// TIA Portal V19 program export: 1 tag tables, 0 data types, 4 data blocks, 12 code blocks (in call order from the OBs), 14 instance data blocks

VAR_GLOBAL   // PLC tag table "System"
   System_Byte AT %MB1 : Byte;
   FirstScan AT %M1.0 : Bool;
   DiagStatusUpdate AT %M1.1 : Bool;
   AlwaysTRUE AT %M1.2 : Bool;
   AlwaysFALSE AT %M1.3 : Bool;
   Clock_Byte AT %MB0 : Byte;
   Clock_10Hz AT %M0.0 : Bool;
   Clock_5Hz AT %M0.1 : Bool;
   "Clock_2.5Hz" AT %M0.2 : Bool;
   Clock_2Hz AT %M0.3 : Bool;
   "Clock_1.25Hz" AT %M0.4 : Bool;
   Clock_1Hz AT %M0.5 : Bool;
   "Clock_0.625Hz" AT %M0.6 : Bool;
   "Clock_0.5Hz" AT %M0.7 : Bool;
   Tag_1 AT %M10.0 : Bool;
END_VAR

DATA_BLOCK "DB_Parameters"   // DB2
{ S7_Optimized_Access := 'TRUE'; DB_Accessible_From_OPC_UA := 'FALSE' }
// stored: DBAccessibleFromOPCUA false, DBAccessibleFromWebserver false, MemoryReserve 100
   VAR RETAIN
      SensorParameter42B4 { ExternalAccessible := 'False'; ExternalVisible := 'False'; ExternalWritable := 'False'} : "stConfigScaleIntReal";   // Parameter for sensor car body detection (42B4 & 42B3)
      SwitchSensorValue { ExternalAccessible := 'False'; ExternalVisible := 'False'; ExternalWritable := 'False'} : Real := 650.0;   // Level parameter switch for car body detection
      uiSpeedLockEccentric { ExternalAccessible := 'False'; ExternalVisible := 'False'; ExternalWritable := 'False'} : UInt := 50;   // Rotation speed for lock eccentric
      RemoveSandPaperParam { ExternalAccessible := 'False'; ExternalVisible := 'False'; ExternalWritable := 'False'} : "stFerRoboticParam";   // FerRobotic parameter for remove the wor sandpaper
      PickUpSandPaperParam { ExternalAccessible := 'False'; ExternalVisible := 'False'; ExternalWritable := 'False'} : "stFerRoboticParam";   // FerRobotic parameter for pich up a new sandpaper
      FlatnessCtrlParam { ExternalAccessible := 'False'; ExternalVisible := 'False'; ExternalWritable := 'False'} : "stFerRoboticParam";   // FerRobotic paramter for flatness contrl disk planeity
      ConfigGreaseZaxis { ExternalAccessible := 'False'; ExternalVisible := 'False'; ExternalWritable := 'False'} : "stConfigGrease";
      ConfigGreaseXaxis { ExternalAccessible := 'False'; ExternalVisible := 'False'; ExternalWritable := 'False'} : "stConfigGrease";
      ConfigVacuumValve { ExternalAccessible := 'False'; ExternalVisible := 'False'; ExternalWritable := 'False'} : "stConfigActuator";
      tTimeoutGimball { ExternalAccessible := 'False'; ExternalVisible := 'False'; ExternalWritable := 'False'} : Time := T#5S;
      tTimeoutEccentric { ExternalAccessible := 'False'; ExternalVisible := 'False'; ExternalWritable := 'False'} : Time := T#20S;
      rFlatnessStrockPos { ExternalAccessible := 'False'; ExternalVisible := 'False'; ExternalWritable := 'False'} : Real := 23.9;   // FerRobotic strock position for control flatness
      rDeltaFlatnessStrock { ExternalAccessible := 'False'; ExternalVisible := 'False'; ExternalWritable := 'False'} : Real := 0.8;   // Delta maxi for flatness control
      nNbDiskLeft { ExternalAccessible := 'False'; ExternalVisible := 'False'; ExternalWritable := 'False'} : USInt := 2;
      nNbDiskRight { ExternalAccessible := 'False'; ExternalVisible := 'False'; ExternalWritable := 'False'} : USInt := 1;
      rLowLimiteStroke { ExternalAccessible := 'False'; ExternalVisible := 'False'; ExternalWritable := 'False'} : Real := 5.0;
      StrokeTooExtend { ExternalAccessible := 'False'; ExternalVisible := 'False'; ExternalWritable := 'False'} : "stHysteresis";
      StrokeTooRetract { ExternalAccessible := 'False'; ExternalVisible := 'False'; ExternalWritable := 'False'} : "stHysteresis";
   END_VAR
BEGIN
   SensorParameter42B4.nInputMin := 0;
   SensorParameter42B4.nIntputMax := 27648;
   SensorParameter42B4.xUniPolar := TRUE;
   SensorParameter42B4.xReverseValue := TRUE;
   SensorParameter42B4.rOutputMin := 200.0;
   SensorParameter42B4.rOutputMax := 1000.0;
   SensorParameter42B4.rOffsetFixe := 0.0;
   SensorParameter42B4.rOffsetProp := 1.0;
   RemoveSandPaperParam.nSetForceTarget := 20;
   RemoveSandPaperParam.nSetForceZero := 10;
   RemoveSandPaperParam.usiSetTimeRamp := 0;
   RemoveSandPaperParam.uiSetSpeed := 0;
   PickUpSandPaperParam.nSetForceTarget := 100;
   PickUpSandPaperParam.nSetForceZero := 0;
   PickUpSandPaperParam.usiSetTimeRamp := 0;
   PickUpSandPaperParam.uiSetSpeed := 0;
   FlatnessCtrlParam.nSetForceTarget := 20;
   FlatnessCtrlParam.nSetForceZero := 0;
   FlatnessCtrlParam.usiSetTimeRamp := 0;
   FlatnessCtrlParam.uiSetSpeed := 0;
   ConfigGreaseZaxis.uiNbPulsePerKm := 4411;
   ConfigGreaseZaxis.uiKmForGreasing := 32;
   ConfigGreaseZaxis.tTimeEnableGreasePump := T#1M;
   ConfigGreaseZaxis.tTimeoutPxGrease := T#1M;
   ConfigGreaseXaxis.uiNbPulsePerKm := 4411;
   ConfigGreaseXaxis.uiKmForGreasing := 32;
   ConfigGreaseXaxis.tTimeEnableGreasePump := T#2M;
   ConfigGreaseXaxis.tTimeoutPxGrease := T#2M;
   ConfigVacuumValve.xEnaMeasureTimeHome := FALSE;
   ConfigVacuumValve.xEnaMeasureTimeAction := FALSE;
   ConfigVacuumValve.xKeepHomeSolActive := FALSE;
   ConfigVacuumValve.xKeepActionSolActive := TRUE;
   ConfigVacuumValve.xPresHomePxSensor := TRUE;
   ConfigVacuumValve.xPresActionPxSensor := TRUE;
   ConfigVacuumValve.tSwitchingCommand := T#50MS;
   ConfigVacuumValve.tTimeOutHomeSensor := T#8S;
   ConfigVacuumValve.tTimeOutActionSensor := T#8S;
   ConfigVacuumValve.tHomeTime := T#3S;
   ConfigVacuumValve.tActionTime := T#3S;
   ConfigVacuumValve.tFilterPxHome := T#100MS;
   ConfigVacuumValve.tFilterPxAction := T#100MS;
   StrokeTooExtend.rValueOn := 40.0;
   StrokeTooExtend.rValueOff := 35.0;
   StrokeTooRetract.rValueOn := 8.0;
   StrokeTooRetract.rValueOff := 13.0;
END_DATA_BLOCK

DATA_BLOCK "DB_Fault"   // DB90
{ S7_Optimized_Access := 'TRUE'; DB_Accessible_From_OPC_UA := 'FALSE' }
// stored: AutoNumber false, DBAccessibleFromOPCUA false, DBAccessibleFromWebserver false, MemoryReserve 100
   VAR
      tonFeedbackZAxisError { ExternalAccessible := 'False'; ExternalVisible := 'False'; ExternalWritable := 'False'} : TON_TIME;
      tonFautLockZAxis { ExternalAccessible := 'False'; ExternalVisible := 'False'; ExternalWritable := 'False'} : TON_TIME;
      tonFaultUnlockZAxis { ExternalAccessible := 'False'; ExternalVisible := 'False'; ExternalWritable := 'False'} : TON_TIME;
      tonFaultStrokTooRetracted { ExternalAccessible := 'False'; ExternalVisible := 'False'; ExternalWritable := 'False'} : TON_TIME;
   END_VAR
BEGIN
END_DATA_BLOCK

DATA_BLOCK "DBF_Safety"   // DB901, F_DB
{ S7_Optimized_Access := 'TRUE' }
// stored: AutoNumber false
   VAR
      TrueSafety { ExternalAccessible := 'False'; ExternalVisible := 'False'; ExternalWritable := 'False'} : Bool := TRUE;   // Bit de securite toujours vrai
      FalseSafety { ExternalAccessible := 'False'; ExternalVisible := 'False'; ExternalWritable := 'False'} : Bool := FALSE;   // Bit de securite toujours faux
      Reset { ExternalAccessible := 'False'; ExternalVisible := 'False'; ExternalWritable := 'False'} : Bool;   // Bit de reset
      i_FdbZAxisBrake { ExternalAccessible := 'False'; ExternalVisible := 'False'; ExternalWritable := 'False'} : Bool;   // Feedback solenoid valve
      i_ResetFromMaster { ExternalAccessible := 'False'; ExternalVisible := 'False'; ExternalWritable := 'False'} : Bool;   // Reset safety from Master PLC
      i_EStopFromMaster { ExternalAccessible := 'False'; ExternalVisible := 'False'; ExternalWritable := 'False'} : Bool;   // Emergency stop from master PLC
      i_OProtectFromMaster { ExternalAccessible := 'False'; ExternalVisible := 'False'; ExternalWritable := 'False'} : Bool;   // Operator Protection from master PLC
      i_AirSupplyEnabledFromMaster { ExternalAccessible := 'False'; ExternalVisible := 'False'; ExternalWritable := 'False'} : Bool;   // Air pressure enabled from master PLC
      i_StopStrokeLimit { ExternalAccessible := 'False'; ExternalVisible := 'False'; ExternalWritable := 'False'} : Bool;   // Stop Stroke limite
      i_VacuumPumpRunning { ExternalAccessible := 'False'; ExternalVisible := 'False'; ExternalWritable := 'False'} : Bool;   // Vacuum pump is running - Zero Speed detection
      o_UnlockZAxis { ExternalAccessible := 'False'; ExternalVisible := 'False'; ExternalWritable := 'False'} : Bool;   // Unlock Z axis of robot
      o_SafetyEnable { ExternalAccessible := 'False'; ExternalVisible := 'False'; ExternalWritable := 'False'} : Bool;   // Safety enabled to Robot Safemove
      o_ExternalEStopToRobot { ExternalAccessible := 'False'; ExternalVisible := 'False'; ExternalWritable := 'False'} : Bool;   // External emergency stop to Robot Safemove
      o_ExternalOProtectToRobot { ExternalAccessible := 'False'; ExternalVisible := 'False'; ExternalWritable := 'False'} : Bool;   // External operator protection to robot Safemove
      o_EStoptoMaster { ExternalAccessible := 'False'; ExternalVisible := 'False'; ExternalWritable := 'False'} : Bool;   // Internal Emergency stop to master PLC
      o_ReqAirSupplyToMaster { ExternalAccessible := 'False'; ExternalVisible := 'False'; ExternalWritable := 'False'} : Bool;   // Request enable air pressure supply to master PLC
      o_RobotStopperToMaster { ExternalAccessible := 'False'; ExternalVisible := 'False'; ExternalWritable := 'False'} : Bool;   // Robot stopped state to master PLC
      o_PowerOffFerRobotic { ExternalAccessible := 'False'; ExternalVisible := 'False'; ExternalWritable := 'False'} : Bool;   // Power Off 24V Safety for FerRobotic
      xErrorReadFromMaster { ExternalAccessible := 'False'; ExternalVisible := 'False'; ExternalWritable := 'False'} : Bool;   // Error read safety data from Master PLC
      xErrorWriteToMaster { ExternalAccessible := 'False'; ExternalVisible := 'False'; ExternalWritable := 'False'} : Bool;   // Error write safety data to Master PLC
   END_VAR
BEGIN
END_DATA_BLOCK

DATA_BLOCK "DB_ToSafety"   // DB999
{ S7_Optimized_Access := 'TRUE' }
// stored: AutoNumber false, MemoryReserve 100
   VAR
      xReset { ExternalAccessible := 'False'; ExternalVisible := 'False'; ExternalWritable := 'False'} : Bool;   // Commande reset general
      xStopStrokeLimit { ExternalAccessible := 'False'; ExternalVisible := 'False'; ExternalWritable := 'False'} : Bool;   // Stop robot on stroke limit retracted
      xSemiAutomaticMode { ExternalAccessible := 'False'; ExternalVisible := 'False'; ExternalWritable := 'False'} : Bool;
   END_VAR
BEGIN
END_DATA_BLOCK

ORGANIZATION_BLOCK "Main"   // OB1, LAD, ProgramCycle
TITLE = "Main Program Sweep (Cycle)"
{ S7_Optimized_Access := 'TRUE' }
// stored: SetENOAutomatically false
   VAR_INPUT
      Initial_Call : Bool;   // Initial call of this OB
      Remanence : Bool;   // =True, if remanent data are available
   END_VAR
BEGIN

REGION Network 1: Commande reset general
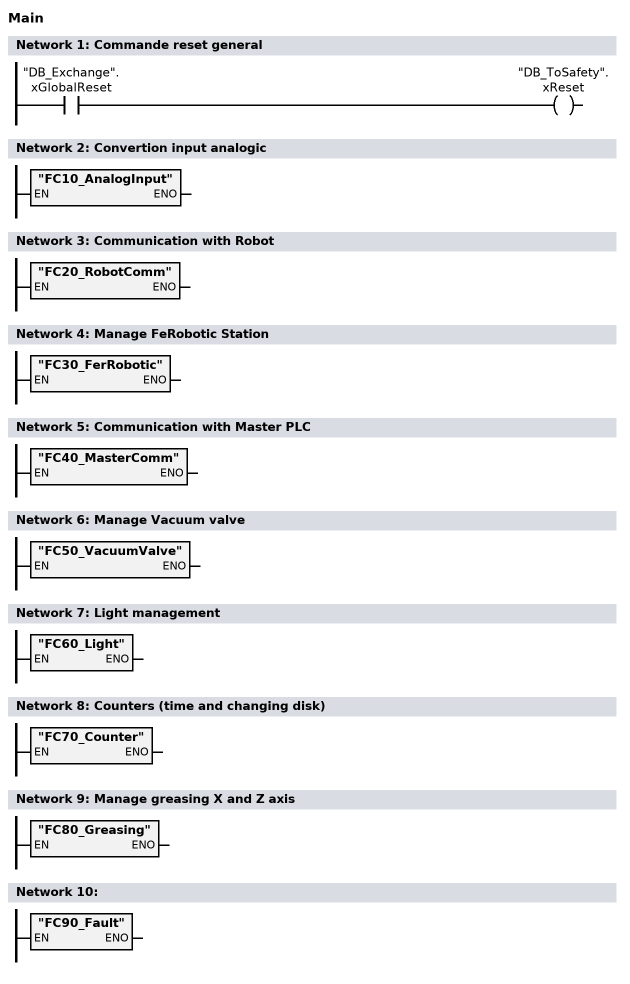
   RUNG wire#powerrail
      Contact( "DB_Exchange".xGlobalReset )
      Coil( "DB_ToSafety".xReset )
   END_RUNG
   // the same network as SCL:
   "DB_ToSafety".xReset := "DB_Exchange".xGlobalReset;
END_REGION

REGION Network 2: Convertion input analogic
   RUNG wire#powerrail
      "FC10_AnalogInput"()
   END_RUNG
   // the same network as SCL:
   "FC10_AnalogInput"();
END_REGION

REGION Network 3: Communication with Robot
   RUNG wire#powerrail
      "FC20_RobotComm"()
   END_RUNG
   // the same network as SCL:
   "FC20_RobotComm"();
END_REGION

REGION Network 4: Manage FeRobotic Station
   RUNG wire#powerrail
      "FC30_FerRobotic"()
   END_RUNG
   // the same network as SCL:
   "FC30_FerRobotic"();
END_REGION

REGION Network 5: Communication with Master PLC
   RUNG wire#powerrail
      "FC40_MasterComm"()
   END_RUNG
   // the same network as SCL:
   "FC40_MasterComm"();
END_REGION

REGION Network 6: Manage Vacuum valve
   RUNG wire#powerrail
      "FC50_VacuumValve"()
   END_RUNG
   // the same network as SCL:
   "FC50_VacuumValve"();
END_REGION

REGION Network 7: Light management
   RUNG wire#powerrail
      "FC60_Light"()
   END_RUNG
   // the same network as SCL:
   "FC60_Light"();
END_REGION

REGION Network 8: Counters (time and changing disk)
   RUNG wire#powerrail
      "FC70_Counter"()
   END_RUNG
   // the same network as SCL:
   "FC70_Counter"();
END_REGION

REGION Network 9: Manage greasing X and Z axis
   RUNG wire#powerrail
      "FC80_Greasing"()
   END_RUNG
   // the same network as SCL:
   "FC80_Greasing"();
END_REGION

REGION Network 10
   RUNG wire#powerrail
      "FC90_Fault"()
   END_RUNG
   // the same network as SCL:
   "FC90_Fault"();
END_REGION
END_ORGANIZATION_BLOCK

FUNCTION "FC30_FerRobotic" : Void   // FC30, LAD
TITLE = FerRobotic communication
{ S7_Optimized_Access := 'TRUE' }
// stored: AutoNumber false, IsIECCheckEnabled true, SetENOAutomatically false
BEGIN

REGION Network 1: Swap byte of value to Receive from FerRobotic
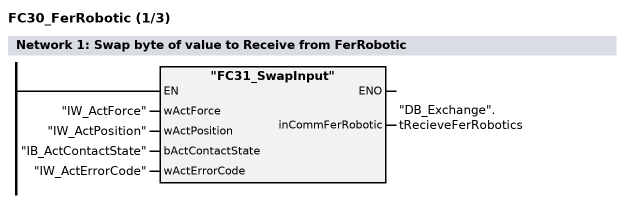
   RUNG wire#powerrail
      "FC31_SwapInput"(wActForce := "IW_ActForce", wActPosition := "IW_ActPosition", bActContactState := "IB_ActContactState", wActErrorCode := "IW_ActErrorCode", inCommFerRobotic => "DB_Exchange".tRecieveFerRobotics)
   END_RUNG
   // the same network as SCL:
   "FC31_SwapInput"(wActForce := "IW_ActForce",
                    wActPosition := "IW_ActPosition",
                    bActContactState := "IB_ActContactState",
                    wActErrorCode := "IW_ActErrorCode",
                    inCommFerRobotic => "DB_Exchange".tRecieveFerRobotics);
END_REGION

REGION Network 2: Comminucation with FerRobotic System
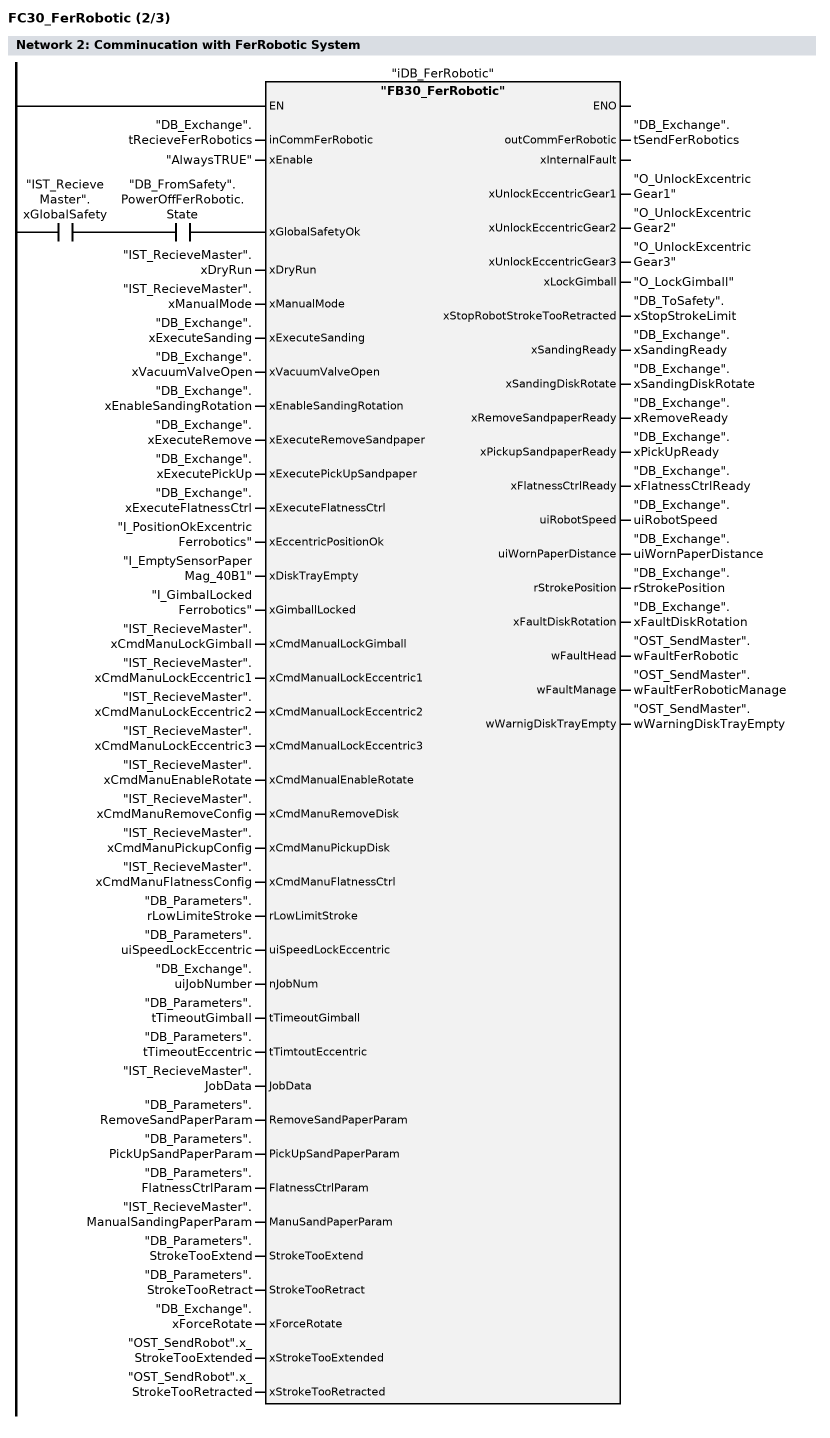
   RUNG wire#powerrail
      "iDB_FerRobotic"(xGlobalSafetyOk := wire#w1, inCommFerRobotic := "DB_Exchange".tRecieveFerRobotics, xEnable := "AlwaysTRUE", xDryRun := "IST_RecieveMaster".xDryRun, xManualMode := "IST_RecieveMaster".xManualMode, xExecuteSanding := "DB_Exchange".xExecuteSanding, xVacuumValveOpen := "DB_Exchange".xVacuumValveOpen, xEnableSandingRotation := "DB_Exchange".xEnableSandingRotation, xExecuteRemoveSandpaper := "DB_Exchange".xExecuteRemove, xExecutePickUpSandpaper := "DB_Exchange".xExecutePickUp, xExecuteFlatnessCtrl := "DB_Exchange".xExecuteFlatnessCtrl, xEccentricPositionOk := "I_PositionOkExcentricFerrobotics", xDiskTrayEmpty := "I_EmptySensorPaperMag_40B1", xGimballLocked := "I_GimbalLockedFerrobotics", xCmdManualLockGimball := "IST_RecieveMaster".xCmdManuLockGimball, xCmdManualLockEccentric1 := "IST_RecieveMaster".xCmdManuLockEccentric1, xCmdManualLockEccentric2 := "IST_RecieveMaster".xCmdManuLockEccentric2, xCmdManualLockEccentric3 := "IST_RecieveMaster".xCmdManuLockEccentric3, xCmdManualEnableRotate := "IST_RecieveMaster".xCmdManuEnableRotate, xCmdManuRemoveDisk := "IST_RecieveMaster".xCmdManuRemoveConfig, xCmdManuPickupDisk := "IST_RecieveMaster".xCmdManuPickupConfig, xCmdManuFlatnessCtrl := "IST_RecieveMaster".xCmdManuFlatnessConfig, rLowLimitStroke := "DB_Parameters".rLowLimiteStroke, uiSpeedLockEccentric := "DB_Parameters".uiSpeedLockEccentric, nJobNum := "DB_Exchange".uiJobNumber, tTimeoutGimball := "DB_Parameters".tTimeoutGimball, tTimtoutEccentric := "DB_Parameters".tTimeoutEccentric, JobData := "IST_RecieveMaster".JobData, RemoveSandPaperParam := "DB_Parameters".RemoveSandPaperParam, PickUpSandPaperParam := "DB_Parameters".PickUpSandPaperParam, FlatnessCtrlParam := "DB_Parameters".FlatnessCtrlParam, ManuSandPaperParam := "IST_RecieveMaster".ManualSandingPaperParam, StrokeTooExtend := "DB_Parameters".StrokeTooExtend, StrokeTooRetract := "DB_Parameters".StrokeTooRetract, xForceRotate := "DB_Exchange".xForceRotate, xStrokeTooExtended := "OST_SendRobot".x_StrokeTooExtended, xStrokeTooRetracted := "OST_SendRobot".x_StrokeTooRetracted, outCommFerRobotic => "DB_Exchange".tSendFerRobotics, xInternalFault =>, xUnlockEccentricGear1 => "O_UnlockExcentricGear1", xUnlockEccentricGear2 => "O_UnlockExcentricGear2", xUnlockEccentricGear3 => "O_UnlockExcentricGear3", xLockGimball => "O_LockGimball", xStopRobotStrokeTooRetracted => "DB_ToSafety".xStopStrokeLimit, xSandingReady => "DB_Exchange".xSandingReady, xSandingDiskRotate => "DB_Exchange".xSandingDiskRotate, xRemoveSandpaperReady => "DB_Exchange".xRemoveReady, xPickupSandpaperReady => "DB_Exchange".xPickUpReady, xFlatnessCtrlReady => "DB_Exchange".xFlatnessCtrlReady, uiRobotSpeed => "DB_Exchange".uiRobotSpeed, uiWornPaperDistance => "DB_Exchange".uiWornPaperDistance, rStrokePosition => "DB_Exchange".rStrokePosition, xFaultDiskRotation => "DB_Exchange".xFaultDiskRotation, wFaultHead => "OST_SendMaster".wFaultFerRobotic, wFaultManage => "OST_SendMaster".wFaultFerRoboticManage, wWarnigDiskTrayEmpty => "OST_SendMaster".wWarningDiskTrayEmpty)
   END_RUNG
   RUNG wire#powerrail
      Contact( "IST_RecieveMaster".xGlobalSafety )
      Contact( "DB_FromSafety".PowerOffFerRobotic.State )
   END_RUNG wire#w1
   // the same network as SCL:
   "iDB_FerRobotic"(inCommFerRobotic := "DB_Exchange".tRecieveFerRobotics,   // "FB30_FerRobotic"
                    xEnable := "AlwaysTRUE",
                    xGlobalSafetyOk := "IST_RecieveMaster".xGlobalSafety AND "DB_FromSafety".PowerOffFerRobotic.State,
                    xDryRun := "IST_RecieveMaster".xDryRun,
                    xManualMode := "IST_RecieveMaster".xManualMode,
                    xExecuteSanding := "DB_Exchange".xExecuteSanding,
                    xVacuumValveOpen := "DB_Exchange".xVacuumValveOpen,
                    xEnableSandingRotation := "DB_Exchange".xEnableSandingRotation,
                    xExecuteRemoveSandpaper := "DB_Exchange".xExecuteRemove,
                    xExecutePickUpSandpaper := "DB_Exchange".xExecutePickUp,
                    xExecuteFlatnessCtrl := "DB_Exchange".xExecuteFlatnessCtrl,
                    xEccentricPositionOk := "I_PositionOkExcentricFerrobotics",
                    xDiskTrayEmpty := "I_EmptySensorPaperMag_40B1",
                    xGimballLocked := "I_GimbalLockedFerrobotics",
                    xCmdManualLockGimball := "IST_RecieveMaster".xCmdManuLockGimball,
                    xCmdManualLockEccentric1 := "IST_RecieveMaster".xCmdManuLockEccentric1,
                    xCmdManualLockEccentric2 := "IST_RecieveMaster".xCmdManuLockEccentric2,
                    xCmdManualLockEccentric3 := "IST_RecieveMaster".xCmdManuLockEccentric3,
                    xCmdManualEnableRotate := "IST_RecieveMaster".xCmdManuEnableRotate,
                    xCmdManuRemoveDisk := "IST_RecieveMaster".xCmdManuRemoveConfig,
                    xCmdManuPickupDisk := "IST_RecieveMaster".xCmdManuPickupConfig,
                    xCmdManuFlatnessCtrl := "IST_RecieveMaster".xCmdManuFlatnessConfig,
                    rLowLimitStroke := "DB_Parameters".rLowLimiteStroke,
                    uiSpeedLockEccentric := "DB_Parameters".uiSpeedLockEccentric,
                    nJobNum := "DB_Exchange".uiJobNumber,
                    tTimeoutGimball := "DB_Parameters".tTimeoutGimball,
                    tTimtoutEccentric := "DB_Parameters".tTimeoutEccentric,
                    JobData := "IST_RecieveMaster".JobData,
                    RemoveSandPaperParam := "DB_Parameters".RemoveSandPaperParam,
                    PickUpSandPaperParam := "DB_Parameters".PickUpSandPaperParam,
                    FlatnessCtrlParam := "DB_Parameters".FlatnessCtrlParam,
                    ManuSandPaperParam := "IST_RecieveMaster".ManualSandingPaperParam,
                    StrokeTooExtend := "DB_Parameters".StrokeTooExtend,
                    StrokeTooRetract := "DB_Parameters".StrokeTooRetract,
                    xForceRotate := "DB_Exchange".xForceRotate,
                    xStrokeTooExtended := "OST_SendRobot".x_StrokeTooExtended,
                    xStrokeTooRetracted := "OST_SendRobot".x_StrokeTooRetracted,
                    outCommFerRobotic => "DB_Exchange".tSendFerRobotics,
                    xUnlockEccentricGear1 => "O_UnlockExcentricGear1",
                    xUnlockEccentricGear2 => "O_UnlockExcentricGear2",
                    xUnlockEccentricGear3 => "O_UnlockExcentricGear3",
                    xLockGimball => "O_LockGimball",
                    xStopRobotStrokeTooRetracted => "DB_ToSafety".xStopStrokeLimit,
                    xSandingReady => "DB_Exchange".xSandingReady,
                    xSandingDiskRotate => "DB_Exchange".xSandingDiskRotate,
                    xRemoveSandpaperReady => "DB_Exchange".xRemoveReady,
                    xPickupSandpaperReady => "DB_Exchange".xPickUpReady,
                    xFlatnessCtrlReady => "DB_Exchange".xFlatnessCtrlReady,
                    uiRobotSpeed => "DB_Exchange".uiRobotSpeed,
                    uiWornPaperDistance => "DB_Exchange".uiWornPaperDistance,
                    rStrokePosition => "DB_Exchange".rStrokePosition,
                    xFaultDiskRotation => "DB_Exchange".xFaultDiskRotation,
                    wFaultHead => "OST_SendMaster".wFaultFerRobotic,
                    wFaultManage => "OST_SendMaster".wFaultFerRoboticManage,
                    wWarnigDiskTrayEmpty => "OST_SendMaster".wWarningDiskTrayEmpty);
END_REGION

REGION Network 3: Swap byte of value to send to FerRobotic
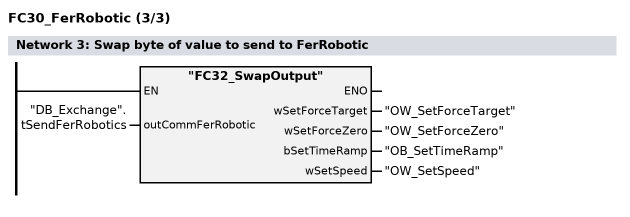
   RUNG wire#powerrail
      "FC32_SwapOutput"(outCommFerRobotic := "DB_Exchange".tSendFerRobotics, wSetForceTarget => "OW_SetForceTarget", wSetForceZero => "OW_SetForceZero", bSetTimeRamp => "OB_SetTimeRamp", wSetSpeed => "OW_SetSpeed")
   END_RUNG
   // the same network as SCL:
   "FC32_SwapOutput"(outCommFerRobotic := "DB_Exchange".tSendFerRobotics,
                     wSetForceTarget => "OW_SetForceTarget",
                     wSetForceZero => "OW_SetForceZero",
                     bSetTimeRamp => "OB_SetTimeRamp",
                     wSetSpeed => "OW_SetSpeed");
END_REGION
END_FUNCTION

FUNCTION "FC31_SwapInput" : Void
{ S7_Optimized_Access := 'TRUE' }
VERSION : 0.1
   VAR_INPUT 
      wActForce : Word;
      wActPosition : Word;
      bActContactState : Byte;
      wActErrorCode : Word;
   END_VAR

   VAR_OUTPUT 
      inCommFerRobotic : "stRecieveFerRobotics";
   END_VAR


BEGIN
	// Swap word of Act Force value
	#inCommFerRobotic.nActForce := WORD_TO_INT( SWAP(#wActForce));
	// Swap word of ActError code value
	#inCommFerRobotic.uiActErrorCode := WORD_TO_UINT(SWAP(#wActErrorCode));
	// Swap word of Act position value
	#inCommFerRobotic.uiActPosition := WORD_TO_UINT(SWAP(#wActPosition));
	// Convert Usint to word of contact state
	#inCommFerRobotic.usiActContactState := BYTE_TO_USINT(#bActContactState);
	
END_FUNCTION

FUNCTION "FC32_SwapOutput" : Void
{ S7_Optimized_Access := 'TRUE' }
VERSION : 0.1
   VAR_INPUT 
      outCommFerRobotic : "stSendFerRobotics";
   END_VAR

   VAR_OUTPUT 
      wSetForceTarget : Word;
      wSetForceZero : Word;
      bSetTimeRamp : Byte;
      wSetSpeed : Word;
   END_VAR


BEGIN
	// Swap word of Set Force Target value
	#wSetForceTarget := SWAP(INT_TO_WORD(#outCommFerRobotic.nSetForceTarget));
	// Swap word of Set Force Zero value
	#wSetForceZero := SWAP(INT_TO_WORD(#outCommFerRobotic.nSetForceZero));
	// Swap word of Set Speed value
	#wSetSpeed := SWAP(UINT_TO_WORD(#outCommFerRobotic.uiSetSpeed));
	// Convert word to USint for time Ramp value
	#bSetTimeRamp := USINT_TO_BYTE(#outCommFerRobotic.usiSetTimeRamp);
	
END_FUNCTION

FUNCTION "FC40_MasterComm" : Void   // FC40, LAD
{ S7_Optimized_Access := 'TRUE' }
// stored: AutoNumber false, IsIECCheckEnabled true, SetENOAutomatically true
BEGIN

REGION Network 1: Master Communication
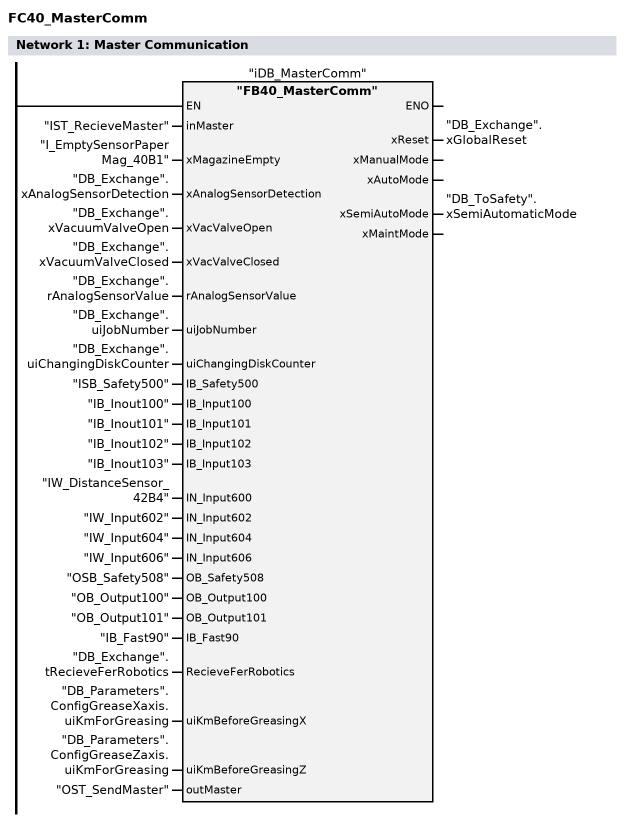
   RUNG wire#powerrail
      "iDB_MasterComm"(inMaster := "IST_RecieveMaster", xMagazineEmpty := "I_EmptySensorPaperMag_40B1", xAnalogSensorDetection := "DB_Exchange".xAnalogSensorDetection, xVacValveOpen := "DB_Exchange".xVacuumValveOpen, xVacValveClosed := "DB_Exchange".xVacuumValveClosed, rAnalogSensorValue := "DB_Exchange".rAnalogSensorValue, uiJobNumber := "DB_Exchange".uiJobNumber, uiChangingDiskCounter := "DB_Exchange".uiChangingDiskCounter, IB_Safety500 := "ISB_Safety500", IB_Input100 := "IB_Inout100", IB_Input101 := "IB_Inout101", IB_Input102 := "IB_Inout102", IB_Input103 := "IB_Inout103", IN_Input600 := "IW_DistanceSensor_42B4", IN_Input602 := "IW_Input602", IN_Input604 := "IW_Input604", IN_Input606 := "IW_Input606", OB_Safety508 := "OSB_Safety508", OB_Output100 := "OB_Output100", OB_Output101 := "OB_Output101", IB_Fast90 := "IB_Fast90", RecieveFerRobotics := "DB_Exchange".tRecieveFerRobotics, uiKmBeforeGreasingX := "DB_Parameters".ConfigGreaseXaxis.uiKmForGreasing, uiKmBeforeGreasingZ := "DB_Parameters".ConfigGreaseZaxis.uiKmForGreasing, outMaster := "OST_SendMaster", xReset => "DB_Exchange".xGlobalReset, xManualMode =>, xAutoMode =>, xSemiAutoMode => "DB_ToSafety".xSemiAutomaticMode, xMaintMode =>)
   END_RUNG
   // the same network as SCL:
   "iDB_MasterComm"(inMaster := "IST_RecieveMaster",   // "FB40_MasterComm"
                    xMagazineEmpty := "I_EmptySensorPaperMag_40B1",
                    xAnalogSensorDetection := "DB_Exchange".xAnalogSensorDetection,
                    xVacValveOpen := "DB_Exchange".xVacuumValveOpen,
                    xVacValveClosed := "DB_Exchange".xVacuumValveClosed,
                    rAnalogSensorValue := "DB_Exchange".rAnalogSensorValue,
                    uiJobNumber := "DB_Exchange".uiJobNumber,
                    uiChangingDiskCounter := "DB_Exchange".uiChangingDiskCounter,
                    IB_Safety500 := "ISB_Safety500",
                    IB_Input100 := "IB_Inout100",
                    IB_Input101 := "IB_Inout101",
                    IB_Input102 := "IB_Inout102",
                    IB_Input103 := "IB_Inout103",
                    IN_Input600 := "IW_DistanceSensor_42B4",
                    IN_Input602 := "IW_Input602",
                    IN_Input604 := "IW_Input604",
                    IN_Input606 := "IW_Input606",
                    OB_Safety508 := "OSB_Safety508",
                    OB_Output100 := "OB_Output100",
                    OB_Output101 := "OB_Output101",
                    IB_Fast90 := "IB_Fast90",
                    RecieveFerRobotics := "DB_Exchange".tRecieveFerRobotics,
                    uiKmBeforeGreasingX := "DB_Parameters".ConfigGreaseXaxis.uiKmForGreasing,
                    uiKmBeforeGreasingZ := "DB_Parameters".ConfigGreaseZaxis.uiKmForGreasing,
                    outMaster := "OST_SendMaster",
                    xReset => "DB_Exchange".xGlobalReset,
                    xSemiAutoMode => "DB_ToSafety".xSemiAutomaticMode);
END_REGION
END_FUNCTION

FUNCTION "FC70_Counter" : Void   // FC2, LAD
{ S7_Optimized_Access := 'TRUE' }
// stored: IsIECCheckEnabled true, SetENOAutomatically false
BEGIN

REGION Network 1: Running time counter
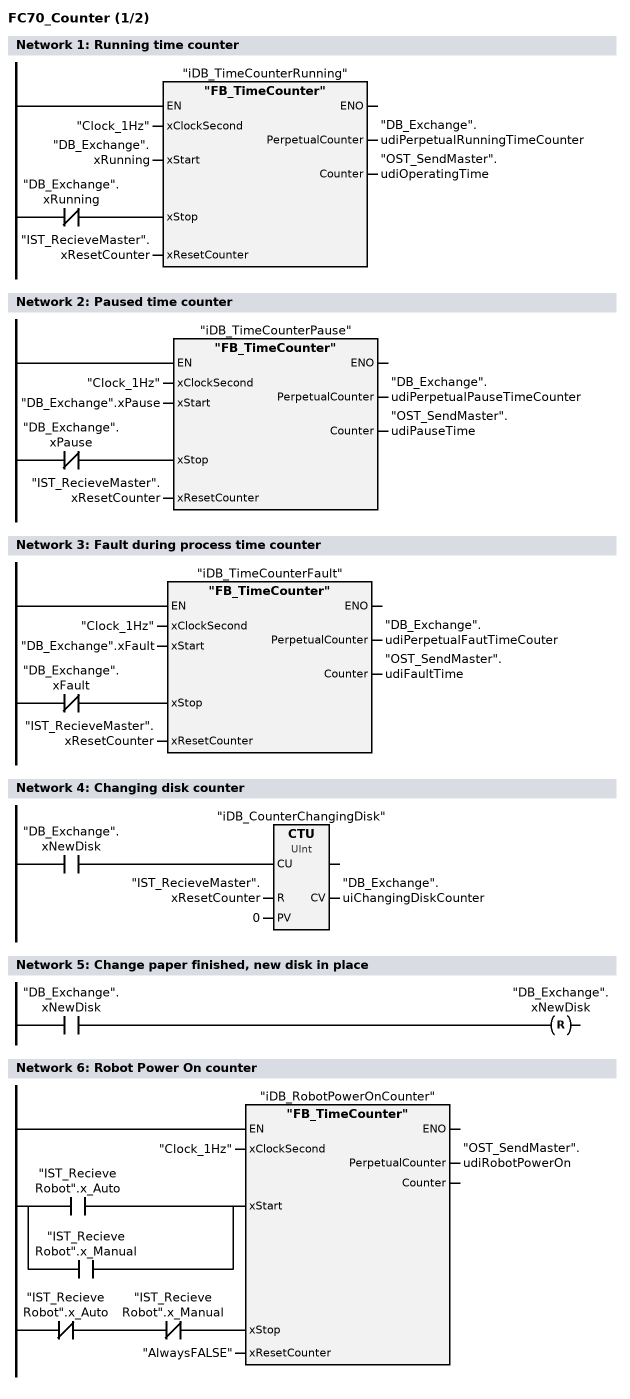
   RUNG wire#powerrail
      "iDB_TimeCounterRunning"(xStop := wire#w1, xClockSecond := "Clock_1Hz", xStart := "DB_Exchange".xRunning, xResetCounter := "IST_RecieveMaster".xResetCounter, PerpetualCounter => "DB_Exchange".udiPerpetualRunningTimeCounter, "Counter" => "OST_SendMaster".udiOperatingTime)
   END_RUNG
   RUNG wire#powerrail
      I_Contact( "DB_Exchange".xRunning )
   END_RUNG wire#w1
   // the same network as SCL:
   "iDB_TimeCounterRunning"(xClockSecond := "Clock_1Hz",   // "FB_TimeCounter"
                           xStart := "DB_Exchange".xRunning,
                           xStop := NOT "DB_Exchange".xRunning,
                           xResetCounter := "IST_RecieveMaster".xResetCounter,
                           PerpetualCounter => "DB_Exchange".udiPerpetualRunningTimeCounter,
                           "Counter" => "OST_SendMaster".udiOperatingTime);
END_REGION

REGION Network 2: Paused time counter
   RUNG wire#powerrail
      "iDB_TimeCounterPause"(xStop := wire#w1, xClockSecond := "Clock_1Hz", xStart := "DB_Exchange".xPause, xResetCounter := "IST_RecieveMaster".xResetCounter, PerpetualCounter => "DB_Exchange".udiPerpetualPauseTimeCounter, "Counter" => "OST_SendMaster".udiPauseTime)
   END_RUNG
   RUNG wire#powerrail
      I_Contact( "DB_Exchange".xPause )
   END_RUNG wire#w1
   // the same network as SCL:
   "iDB_TimeCounterPause"(xClockSecond := "Clock_1Hz",   // "FB_TimeCounter"
                          xStart := "DB_Exchange".xPause,
                          xStop := NOT "DB_Exchange".xPause,
                          xResetCounter := "IST_RecieveMaster".xResetCounter,
                          PerpetualCounter => "DB_Exchange".udiPerpetualPauseTimeCounter,
                          "Counter" => "OST_SendMaster".udiPauseTime);
END_REGION

REGION Network 3: Fault during process time counter
   RUNG wire#powerrail
      "iDB_TimeCounterFault"(xStop := wire#w1, xClockSecond := "Clock_1Hz", xStart := "DB_Exchange".xFault, xResetCounter := "IST_RecieveMaster".xResetCounter, PerpetualCounter => "DB_Exchange".udiPerpetualFautTimeCouter, "Counter" => "OST_SendMaster".udiFaultTime)
   END_RUNG
   RUNG wire#powerrail
      I_Contact( "DB_Exchange".xFault )
   END_RUNG wire#w1
   // the same network as SCL:
   "iDB_TimeCounterFault"(xClockSecond := "Clock_1Hz",   // "FB_TimeCounter"
                          xStart := "DB_Exchange".xFault,
                          xStop := NOT "DB_Exchange".xFault,
                          xResetCounter := "IST_RecieveMaster".xResetCounter,
                          PerpetualCounter => "DB_Exchange".udiPerpetualFautTimeCouter,
                          "Counter" => "OST_SendMaster".udiFaultTime);
END_REGION

REGION Network 4: Changing disk counter
   RUNG wire#powerrail
      Contact( "DB_Exchange".xNewDisk )
      { S7_Templates := "value_type := UInt" } "iDB_CounterChangingDisk".CTU(r := "IST_RecieveMaster".xResetCounter, pv := 0, cv => "DB_Exchange".uiChangingDiskCounter)
   END_RUNG
   // the same network as SCL:
   "iDB_CounterChangingDisk".CTU(CU := "DB_Exchange".xNewDisk,
                           R := "IST_RecieveMaster".xResetCounter,
                           PV := 0,
                           CV => "DB_Exchange".uiChangingDiskCounter);
END_REGION

REGION Network 5: Change paper finished, new disk in place
   RUNG wire#powerrail
      Contact( "DB_Exchange".xNewDisk )
      R_Coil( "DB_Exchange".xNewDisk )
   END_RUNG
   // the same network as SCL:
   IF "DB_Exchange".xNewDisk THEN "DB_Exchange".xNewDisk := FALSE; END_IF;
END_REGION

REGION Network 6: Robot Power On counter
   RUNG wire#powerrail
      "iDB_RobotPowerOnCounter"(xStart := wire#w1, xStop := wire#w2, xClockSecond := "Clock_1Hz", xResetCounter := "AlwaysFALSE", PerpetualCounter => "OST_SendMaster".udiRobotPowerOn, "Counter" =>)
   END_RUNG
   RUNG wire#powerrail
      Contact( "IST_RecieveRobot".x_Auto )
   END_RUNG wire#w1
   RUNG wire#powerrail
      Contact( "IST_RecieveRobot".x_Manual )
   END_RUNG wire#w1
   RUNG wire#powerrail
      I_Contact( "IST_RecieveRobot".x_Auto )
      I_Contact( "IST_RecieveRobot".x_Manual )
   END_RUNG wire#w2
   // the same network as SCL:
   "iDB_RobotPowerOnCounter"(xClockSecond := "Clock_1Hz",   // "FB_TimeCounter"
                           xStart := "IST_RecieveRobot".x_Auto OR "IST_RecieveRobot".x_Manual,
                           xStop := NOT "IST_RecieveRobot".x_Auto AND NOT "IST_RecieveRobot".x_Manual,
                           xResetCounter := "AlwaysFALSE",
                           PerpetualCounter => "OST_SendMaster".udiRobotPowerOn);
END_REGION

REGION Network 7: Robot Drive On counter
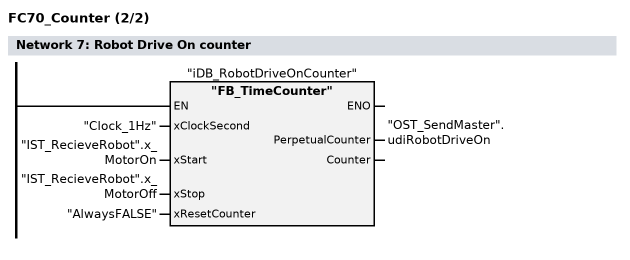
   RUNG wire#powerrail
      "iDB_RobotDriveOnCounter"(xClockSecond := "Clock_1Hz", xStart := "IST_RecieveRobot".x_MotorOn, xStop := "IST_RecieveRobot".x_MotorOff, xResetCounter := "AlwaysFALSE", PerpetualCounter => "OST_SendMaster".udiRobotDriveOn, "Counter" =>)
   END_RUNG
   // the same network as SCL:
   "iDB_RobotDriveOnCounter"(xClockSecond := "Clock_1Hz",   // "FB_TimeCounter"
                           xStart := "IST_RecieveRobot".x_MotorOn,
                           xStop := "IST_RecieveRobot".x_MotorOff,
                           xResetCounter := "AlwaysFALSE",
                           PerpetualCounter => "OST_SendMaster".udiRobotDriveOn);
END_REGION
END_FUNCTION

FUNCTION "FC80_Greasing" : Void   // FC80, LAD
{ S7_Optimized_Access := 'TRUE' }
// stored: AutoNumber false, SetENOAutomatically false
BEGIN

REGION Network 1: Manage greasing X axis
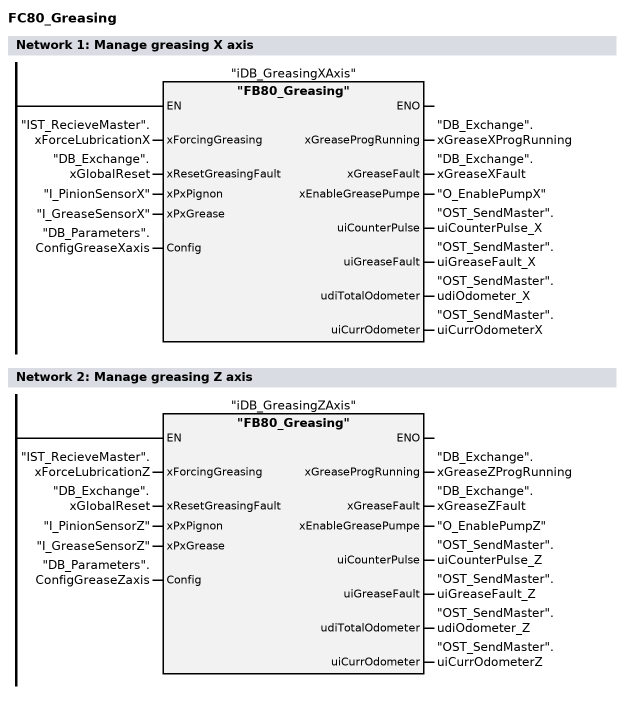
   RUNG wire#powerrail
      "iDB_GreasingXAxis"(xForcingGreasing := "IST_RecieveMaster".xForceLubricationX, xResetGreasingFault := "DB_Exchange".xGlobalReset, xPxPignon := "I_PinionSensorX", xPxGrease := "I_GreaseSensorX", Config := "DB_Parameters".ConfigGreaseXaxis, xGreaseProgRunning => "DB_Exchange".xGreaseXProgRunning, xGreaseFault => "DB_Exchange".xGreaseXFault, xEnableGreasePumpe => "O_EnablePumpX", uiCounterPulse => "OST_SendMaster".uiCounterPulse_X, uiGreaseFault => "OST_SendMaster".uiGreaseFault_X, udiTotalOdometer => "OST_SendMaster".udiOdometer_X, uiCurrOdometer => "OST_SendMaster".uiCurrOdometerX)
   END_RUNG
   // the same network as SCL:
   "iDB_GreasingXAxis"(xForcingGreasing := "IST_RecieveMaster".xForceLubricationX,   // "FB80_Greasing"
                       xResetGreasingFault := "DB_Exchange".xGlobalReset,
                       xPxPignon := "I_PinionSensorX",
                       xPxGrease := "I_GreaseSensorX",
                       Config := "DB_Parameters".ConfigGreaseXaxis,
                       xGreaseProgRunning => "DB_Exchange".xGreaseXProgRunning,
                       xGreaseFault => "DB_Exchange".xGreaseXFault,
                       xEnableGreasePumpe => "O_EnablePumpX",
                       uiCounterPulse => "OST_SendMaster".uiCounterPulse_X,
                       uiGreaseFault => "OST_SendMaster".uiGreaseFault_X,
                       udiTotalOdometer => "OST_SendMaster".udiOdometer_X,
                       uiCurrOdometer => "OST_SendMaster".uiCurrOdometerX);
END_REGION

REGION Network 2: Manage greasing Z axis
   RUNG wire#powerrail
      "iDB_GreasingZAxis"(xForcingGreasing := "IST_RecieveMaster".xForceLubricationZ, xResetGreasingFault := "DB_Exchange".xGlobalReset, xPxPignon := "I_PinionSensorZ", xPxGrease := "I_GreaseSensorZ", Config := "DB_Parameters".ConfigGreaseZaxis, xGreaseProgRunning => "DB_Exchange".xGreaseZProgRunning, xGreaseFault => "DB_Exchange".xGreaseZFault, xEnableGreasePumpe => "O_EnablePumpZ", uiCounterPulse => "OST_SendMaster".uiCounterPulse_Z, uiGreaseFault => "OST_SendMaster".uiGreaseFault_Z, udiTotalOdometer => "OST_SendMaster".udiOdometer_Z, uiCurrOdometer => "OST_SendMaster".uiCurrOdometerZ)
   END_RUNG
   // the same network as SCL:
   "iDB_GreasingZAxis"(xForcingGreasing := "IST_RecieveMaster".xForceLubricationZ,   // "FB80_Greasing"
                       xResetGreasingFault := "DB_Exchange".xGlobalReset,
                       xPxPignon := "I_PinionSensorZ",
                       xPxGrease := "I_GreaseSensorZ",
                       Config := "DB_Parameters".ConfigGreaseZaxis,
                       xGreaseProgRunning => "DB_Exchange".xGreaseZProgRunning,
                       xGreaseFault => "DB_Exchange".xGreaseZFault,
                       xEnableGreasePumpe => "O_EnablePumpZ",
                       uiCounterPulse => "OST_SendMaster".uiCounterPulse_Z,
                       uiGreaseFault => "OST_SendMaster".uiGreaseFault_Z,
                       udiTotalOdometer => "OST_SendMaster".udiOdometer_Z,
                       uiCurrOdometer => "OST_SendMaster".uiCurrOdometerZ);
END_REGION
END_FUNCTION

FUNCTION "FC90_Fault" : Void   // FC90, LAD
{ S7_Optimized_Access := 'TRUE' }
// stored: AutoNumber false, IsIECCheckEnabled true, SetENOAutomatically false
BEGIN

REGION Network 1: Fault no manage by function
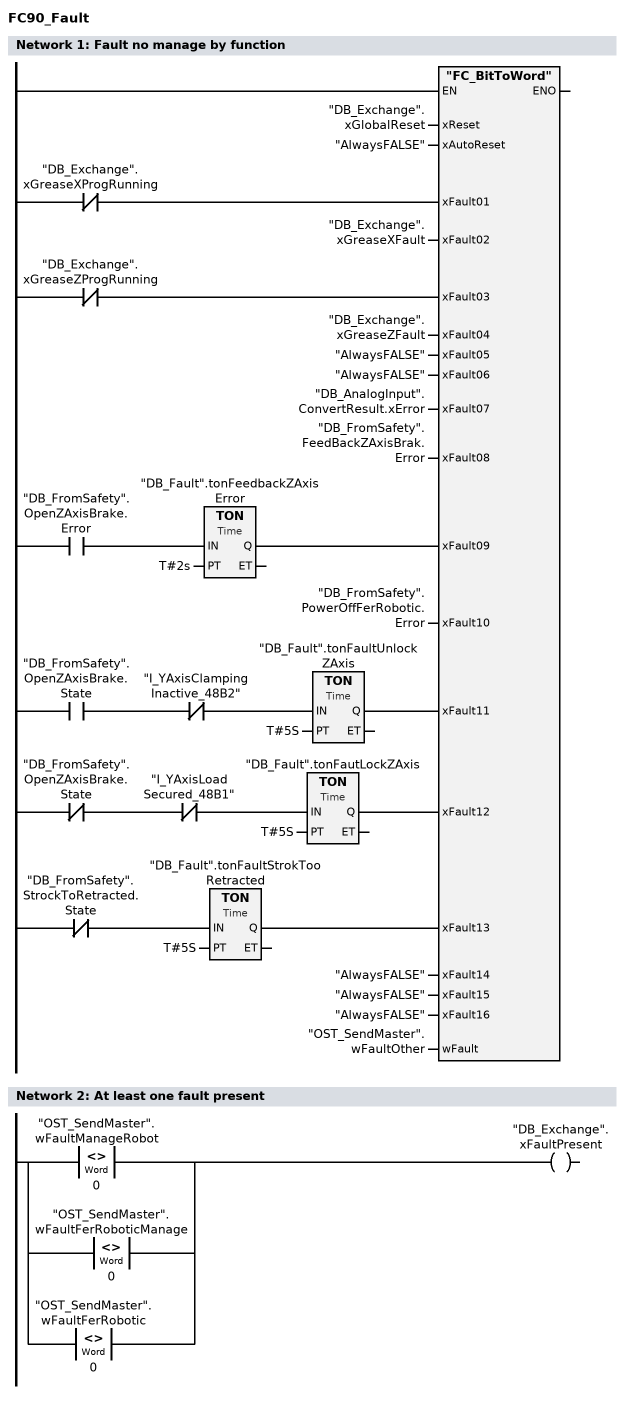
   RUNG wire#powerrail
      "FC_BitToWord"(xFault01 := wire#w1, xFault03 := wire#w2, xFault09 := wire#w3, xFault11 := wire#w4, xFault12 := wire#w5, xFault13 := wire#w6, xReset := "DB_Exchange".xGlobalReset, xAutoReset := "AlwaysFALSE", xFault02 := "DB_Exchange".xGreaseXFault, xFault04 := "DB_Exchange".xGreaseZFault, xFault05 := "AlwaysFALSE", xFault06 := "AlwaysFALSE", xFault07 := "DB_AnalogInput".ConvertResult.xError, xFault08 := "DB_FromSafety".FeedBackZAxisBrak.Error, xFault10 := "DB_FromSafety".PowerOffFerRobotic.Error, xFault14 := "AlwaysFALSE", xFault15 := "AlwaysFALSE", xFault16 := "AlwaysFALSE", wFault := "OST_SendMaster".wFaultOther)
   END_RUNG
   RUNG wire#powerrail
      I_Contact( "DB_Exchange".xGreaseXProgRunning )
   END_RUNG wire#w1
   RUNG wire#powerrail
      I_Contact( "DB_Exchange".xGreaseZProgRunning )
   END_RUNG wire#w2
   RUNG wire#powerrail
      Contact( "DB_FromSafety".OpenZAxisBrake.Error )
      { S7_Templates := "time_type := Time" } "DB_Fault".tonFeedbackZAxisError.TON(pt := T#2s, et =>)
   END_RUNG wire#w3
   RUNG wire#powerrail
      Contact( "DB_FromSafety".OpenZAxisBrake.State )
      I_Contact( "I_YAxisClampingInactive_48B2" )
      { S7_Templates := "time_type := Time" } "DB_Fault".tonFaultUnlockZAxis.TON(pt := T#5S, et =>)
   END_RUNG wire#w4
   RUNG wire#powerrail
      I_Contact( "DB_FromSafety".OpenZAxisBrake.State )
      I_Contact( "I_YAxisLoadSecured_48B1" )
      { S7_Templates := "time_type := Time" } "DB_Fault".tonFautLockZAxis.TON(pt := T#5S, et =>)
   END_RUNG wire#w5
   RUNG wire#powerrail
      I_Contact( "DB_FromSafety".StrockToRetracted.State )
      { S7_Templates := "time_type := Time" } "DB_Fault".tonFaultStrokTooRetracted.TON(pt := T#5S, et =>)
   END_RUNG wire#w6
   // the same network as SCL:
   "DB_Fault".tonFeedbackZAxisError.TON(IN := "DB_FromSafety".OpenZAxisBrake.Error, PT := T#2s);
   "DB_Fault".tonFaultUnlockZAxis.TON(IN := "DB_FromSafety".OpenZAxisBrake.State AND NOT "I_YAxisClampingInactive_48B2",
                           PT := T#5S);
   "DB_Fault".tonFautLockZAxis.TON(IN := NOT "DB_FromSafety".OpenZAxisBrake.State AND NOT "I_YAxisLoadSecured_48B1",
                           PT := T#5S);
   "DB_Fault".tonFaultStrokTooRetracted.TON(IN := NOT "DB_FromSafety".StrockToRetracted.State, PT := T#5S);
   "FC_BitToWord"(xReset := "DB_Exchange".xGlobalReset,
                  xAutoReset := "AlwaysFALSE",
                  xFault01 := NOT "DB_Exchange".xGreaseXProgRunning,
                  xFault02 := "DB_Exchange".xGreaseXFault,
                  xFault03 := NOT "DB_Exchange".xGreaseZProgRunning,
                  xFault04 := "DB_Exchange".xGreaseZFault,
                  xFault05 := "AlwaysFALSE",
                  xFault06 := "AlwaysFALSE",
                  xFault07 := "DB_AnalogInput".ConvertResult.xError,
                  xFault08 := "DB_FromSafety".FeedBackZAxisBrak.Error,
                  xFault09 := "DB_Fault".tonFeedbackZAxisError.Q,
                  xFault10 := "DB_FromSafety".PowerOffFerRobotic.Error,
                  xFault11 := "DB_Fault".tonFaultUnlockZAxis.Q,
                  xFault12 := "DB_Fault".tonFautLockZAxis.Q,
                  xFault13 := "DB_Fault".tonFaultStrokTooRetracted.Q,
                  xFault14 := "AlwaysFALSE",
                  xFault15 := "AlwaysFALSE",
                  xFault16 := "AlwaysFALSE",
                  wFault := "OST_SendMaster".wFaultOther);
END_REGION

REGION Network 2: At least one fault present
   RUNG wire#powerrail
      { S7_Templates := "SrcType := Word" } NE_Contact(in1 := "OST_SendMaster".wFaultManageRobot, in2 := 0)
      wire#w1
      Coil( "DB_Exchange".xFaultPresent )
   END_RUNG
   RUNG wire#powerrail
      { S7_Templates := "SrcType := Word" } NE_Contact(in1 := "OST_SendMaster".wFaultFerRoboticManage, in2 := 0)
   END_RUNG wire#w1
   RUNG wire#powerrail
      { S7_Templates := "SrcType := Word" } NE_Contact(in1 := "OST_SendMaster".wFaultFerRobotic, in2 := 0)
   END_RUNG wire#w1
   // the same network as SCL:
   "DB_Exchange".xFaultPresent := ("OST_SendMaster".wFaultManageRobot <> 0) OR ("OST_SendMaster".wFaultFerRoboticManage <> 0) OR ("OST_SendMaster".wFaultFerRobotic <> 0);
END_REGION
END_FUNCTION

FUNCTION "FC900_SafetyIntegration" : Void   // FC900, F_LAD
{ S7_Optimized_Access := 'TRUE' }
// stored: AutoNumber false
BEGIN

REGION Network 1: Bit de reset
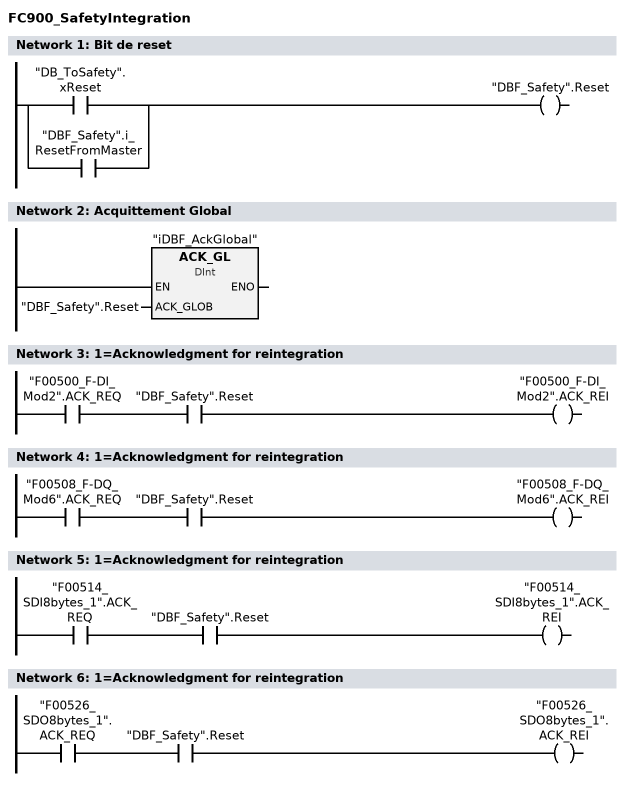
   RUNG wire#powerrail
      Contact( "DB_ToSafety".xReset )
      wire#w1
      Coil( "DBF_Safety".Reset )
   END_RUNG
   RUNG wire#powerrail
      Contact( "DBF_Safety".i_ResetFromMaster )
   END_RUNG wire#w1
   // the same network as SCL:
   "DBF_Safety".Reset := "DB_ToSafety".xReset OR "DBF_Safety".i_ResetFromMaster;
END_REGION

REGION Network 2: Acquittement Global
   RUNG wire#powerrail
      { S7_Templates := "codedbool_type := DInt" } "iDBF_AckGlobal".ACK_GL(ACK_GLOB := "DBF_Safety".Reset)
   END_RUNG
   // the same network as SCL:
   "iDBF_AckGlobal"(ACK_GLOB := "DBF_Safety".Reset);   // ACK_GL
END_REGION

REGION Network 3: 1=Acknowledgment for reintegration
   RUNG wire#powerrail
      Contact( "F00500_F-DI_Mod2".ACK_REQ )
      Contact( "DBF_Safety".Reset )
      Coil( "F00500_F-DI_Mod2".ACK_REI )
   END_RUNG
   // the same network as SCL:
   "F00500_F-DI_Mod2".ACK_REI := "F00500_F-DI_Mod2".ACK_REQ AND "DBF_Safety".Reset;
END_REGION

REGION Network 4: 1=Acknowledgment for reintegration
   RUNG wire#powerrail
      Contact( "F00508_F-DQ_Mod6".ACK_REQ )
      Contact( "DBF_Safety".Reset )
      Coil( "F00508_F-DQ_Mod6".ACK_REI )
   END_RUNG
   // the same network as SCL:
   "F00508_F-DQ_Mod6".ACK_REI := "F00508_F-DQ_Mod6".ACK_REQ AND "DBF_Safety".Reset;
END_REGION

REGION Network 5: 1=Acknowledgment for reintegration
   RUNG wire#powerrail
      Contact( "F00514_SDI8bytes_1".ACK_REQ )
      Contact( "DBF_Safety".Reset )
      Coil( "F00514_SDI8bytes_1".ACK_REI )
   END_RUNG
   // the same network as SCL:
   "F00514_SDI8bytes_1".ACK_REI := "F00514_SDI8bytes_1".ACK_REQ AND "DBF_Safety".Reset;
END_REGION

REGION Network 6: 1=Acknowledgment for reintegration
   RUNG wire#powerrail
      Contact( "F00526_SDO8bytes_1".ACK_REQ )
      Contact( "DBF_Safety".Reset )
      Coil( "F00526_SDO8bytes_1".ACK_REI )
   END_RUNG
   // the same network as SCL:
   "F00526_SDO8bytes_1".ACK_REI := "F00526_SDO8bytes_1".ACK_REQ AND "DBF_Safety".Reset;
END_REGION
END_FUNCTION

FUNCTION "FC901_SafetyInputs" : Void   // FC901, F_LAD
{ S7_Optimized_Access := 'TRUE' }
// stored: AutoNumber false
BEGIN

REGION Network 1: Feedback solenoid valve
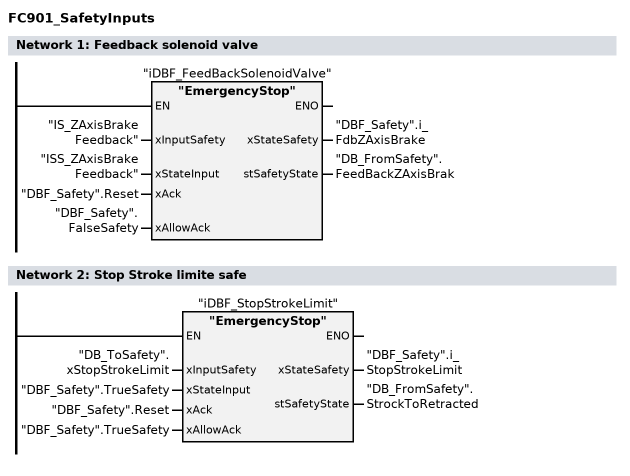
   RUNG wire#powerrail
      "iDBF_FeedBackSolenoidValve"(xInputSafety := "IS_ZAxisBrakeFeedback", xStateInput := "ISS_ZAxisBrakeFeedback", xAck := "DBF_Safety".Reset, xAllowAck := "DBF_Safety".FalseSafety, xStateSafety => "DBF_Safety".i_FdbZAxisBrake, stSafetyState => "DB_FromSafety".FeedBackZAxisBrak)
   END_RUNG
   // the same network as SCL:
   "iDBF_FeedBackSolenoidValve"(xInputSafety := "IS_ZAxisBrakeFeedback",   // "EmergencyStop"
                           xStateInput := "ISS_ZAxisBrakeFeedback",
                           xAck := "DBF_Safety".Reset,
                           xAllowAck := "DBF_Safety".FalseSafety,
                           xStateSafety => "DBF_Safety".i_FdbZAxisBrake,
                           stSafetyState => "DB_FromSafety".FeedBackZAxisBrak);
END_REGION

REGION Network 2: Stop Stroke limite safe
   RUNG wire#powerrail
      "iDBF_StopStrokeLimit"(xInputSafety := "DB_ToSafety".xStopStrokeLimit, xStateInput := "DBF_Safety".TrueSafety, xAck := "DBF_Safety".Reset, xAllowAck := "DBF_Safety".TrueSafety, xStateSafety => "DBF_Safety".i_StopStrokeLimit, stSafetyState => "DB_FromSafety".StrockToRetracted)
   END_RUNG
   // the same network as SCL:
   "iDBF_StopStrokeLimit"(xInputSafety := "DB_ToSafety".xStopStrokeLimit,   // "EmergencyStop"
                          xStateInput := "DBF_Safety".TrueSafety,
                          xAck := "DBF_Safety".Reset,
                          xAllowAck := "DBF_Safety".TrueSafety,
                          xStateSafety => "DBF_Safety".i_StopStrokeLimit,
                          stSafetyState => "DB_FromSafety".StrockToRetracted);
END_REGION
END_FUNCTION

FUNCTION "FC903_SafetyOutputs" : Void   // FC903, F_LAD
{ S7_Optimized_Access := 'TRUE' }
// stored: AutoNumber false
BEGIN

REGION Network 1: Open Z Axis brake
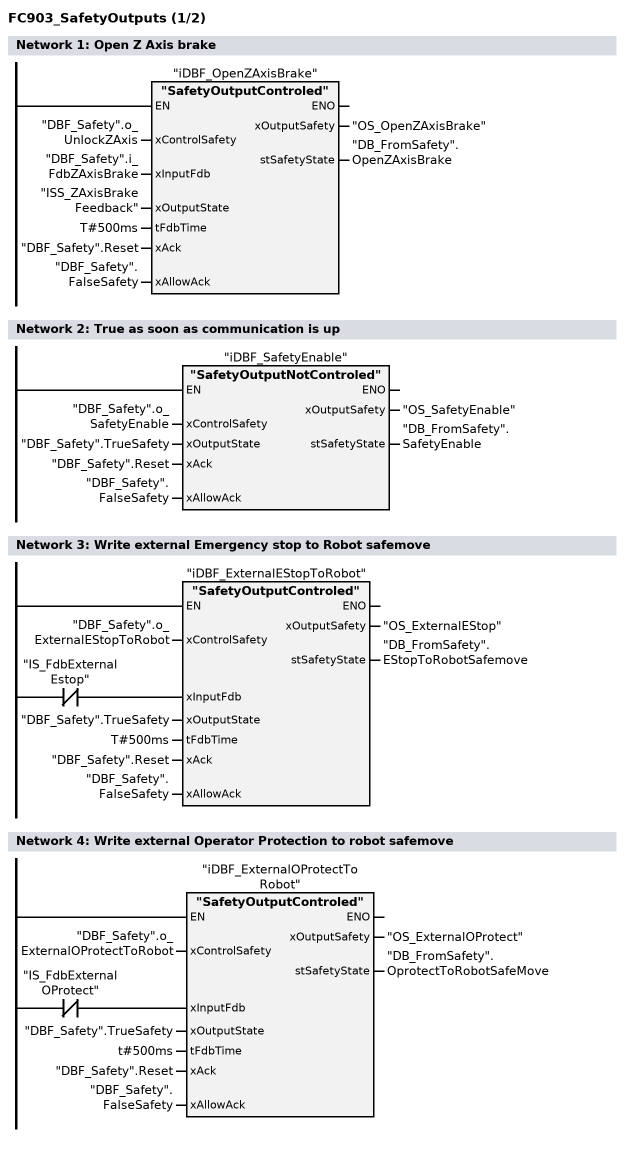
   RUNG wire#powerrail
      "iDBF_OpenZAxisBrake"(xControlSafety := "DBF_Safety".o_UnlockZAxis, xInputFdb := "DBF_Safety".i_FdbZAxisBrake, xOutputState := "ISS_ZAxisBrakeFeedback", tFdbTime := T#500ms, xAck := "DBF_Safety".Reset, xAllowAck := "DBF_Safety".FalseSafety, xOutputSafety => "OS_OpenZAxisBrake", stSafetyState => "DB_FromSafety".OpenZAxisBrake)
   END_RUNG
   // the same network as SCL:
   "iDBF_OpenZAxisBrake"(xControlSafety := "DBF_Safety".o_UnlockZAxis,   // "SafetyOutputControled"
                         xInputFdb := "DBF_Safety".i_FdbZAxisBrake,
                         xOutputState := "ISS_ZAxisBrakeFeedback",
                         tFdbTime := T#500ms,
                         xAck := "DBF_Safety".Reset,
                         xAllowAck := "DBF_Safety".FalseSafety,
                         xOutputSafety => "OS_OpenZAxisBrake",
                         stSafetyState => "DB_FromSafety".OpenZAxisBrake);
END_REGION

REGION Network 2: True as soon as communication is up
   RUNG wire#powerrail
      "iDBF_SafetyEnable"(xControlSafety := "DBF_Safety".o_SafetyEnable, xOutputState := "DBF_Safety".TrueSafety, xAck := "DBF_Safety".Reset, xAllowAck := "DBF_Safety".FalseSafety, xOutputSafety => "OS_SafetyEnable", stSafetyState => "DB_FromSafety".SafetyEnable)
   END_RUNG
   // the same network as SCL:
   "iDBF_SafetyEnable"(xControlSafety := "DBF_Safety".o_SafetyEnable,   // "SafetyOutputNotControled"
                       xOutputState := "DBF_Safety".TrueSafety,
                       xAck := "DBF_Safety".Reset,
                       xAllowAck := "DBF_Safety".FalseSafety,
                       xOutputSafety => "OS_SafetyEnable",
                       stSafetyState => "DB_FromSafety".SafetyEnable);
END_REGION

REGION Network 3: Write external Emergency stop to Robot safemove
   RUNG wire#powerrail
      "iDBF_ExternalEStopToRobot"(xInputFdb := wire#w1, xControlSafety := "DBF_Safety".o_ExternalEStopToRobot, xOutputState := "DBF_Safety".TrueSafety, tFdbTime := T#500ms, xAck := "DBF_Safety".Reset, xAllowAck := "DBF_Safety".FalseSafety, xOutputSafety => "OS_ExternalEStop", stSafetyState => "DB_FromSafety".EStopToRobotSafemove)
   END_RUNG
   RUNG wire#powerrail
      I_Contact( "IS_FdbExternalEstop" )
   END_RUNG wire#w1
   // the same network as SCL:
   "iDBF_ExternalEStopToRobot"(xControlSafety := "DBF_Safety".o_ExternalEStopToRobot,   // "SafetyOutputControled"
                           xInputFdb := NOT "IS_FdbExternalEstop",
                           xOutputState := "DBF_Safety".TrueSafety,
                           tFdbTime := T#500ms,
                           xAck := "DBF_Safety".Reset,
                           xAllowAck := "DBF_Safety".FalseSafety,
                           xOutputSafety => "OS_ExternalEStop",
                           stSafetyState => "DB_FromSafety".EStopToRobotSafemove);
END_REGION

REGION Network 4: Write external Operator Protection to robot safemove
   RUNG wire#powerrail
      "iDBF_ExternalOProtectToRobot"(xInputFdb := wire#w1, xControlSafety := "DBF_Safety".o_ExternalOProtectToRobot, xOutputState := "DBF_Safety".TrueSafety, tFdbTime := t#500ms, xAck := "DBF_Safety".Reset, xAllowAck := "DBF_Safety".FalseSafety, xOutputSafety => "OS_ExternalOProtect", stSafetyState => "DB_FromSafety".OprotectToRobotSafeMove)
   END_RUNG
   RUNG wire#powerrail
      I_Contact( "IS_FdbExternalOProtect" )
   END_RUNG wire#w1
   // the same network as SCL:
   "iDBF_ExternalOProtectToRobot"(xControlSafety := "DBF_Safety".o_ExternalOProtectToRobot,   // "SafetyOutputControled"
                           xInputFdb := NOT "IS_FdbExternalOProtect",
                           xOutputState := "DBF_Safety".TrueSafety,
                           tFdbTime := t#500ms,
                           xAck := "DBF_Safety".Reset,
                           xAllowAck := "DBF_Safety".FalseSafety,
                           xOutputSafety => "OS_ExternalOProtect",
                           stSafetyState => "DB_FromSafety".OprotectToRobotSafeMove);
END_REGION

REGION Network 5: Power Off 24V safety for FerRobotic Head
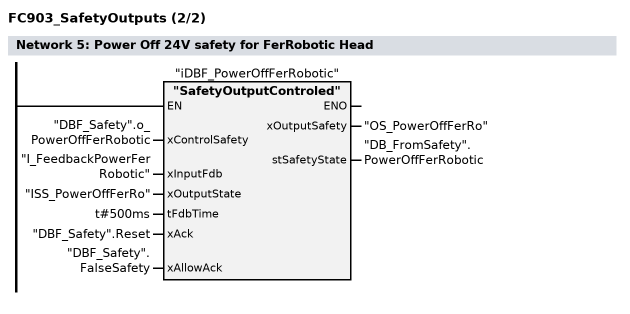
   RUNG wire#powerrail
      "iDBF_PowerOffFerRobotic"(xControlSafety := "DBF_Safety".o_PowerOffFerRobotic, xInputFdb := "I_FeedbackPowerFerRobotic", xOutputState := "ISS_PowerOffFerRo", tFdbTime := t#500ms, xAck := "DBF_Safety".Reset, xAllowAck := "DBF_Safety".FalseSafety, xOutputSafety => "OS_PowerOffFerRo", stSafetyState => "DB_FromSafety".PowerOffFerRobotic)
   END_RUNG
   // the same network as SCL:
   "iDBF_PowerOffFerRobotic"(xControlSafety := "DBF_Safety".o_PowerOffFerRobotic,   // "SafetyOutputControled"
                           xInputFdb := "I_FeedbackPowerFerRobotic",
                           xOutputState := "ISS_PowerOffFerRo",
                           tFdbTime := t#500ms,
                           xAck := "DBF_Safety".Reset,
                           xAllowAck := "DBF_Safety".FalseSafety,
                           xOutputSafety => "OS_PowerOffFerRo",
                           stSafetyState => "DB_FromSafety".PowerOffFerRobotic);
END_REGION
END_FUNCTION

FUNCTION_BLOCK "MainSafety"   // FB900, F_LAD
{ S7_Optimized_Access := 'TRUE' }
// stored: AutoNumber false
BEGIN

REGION Network 1: Read the safety data from Master PLC
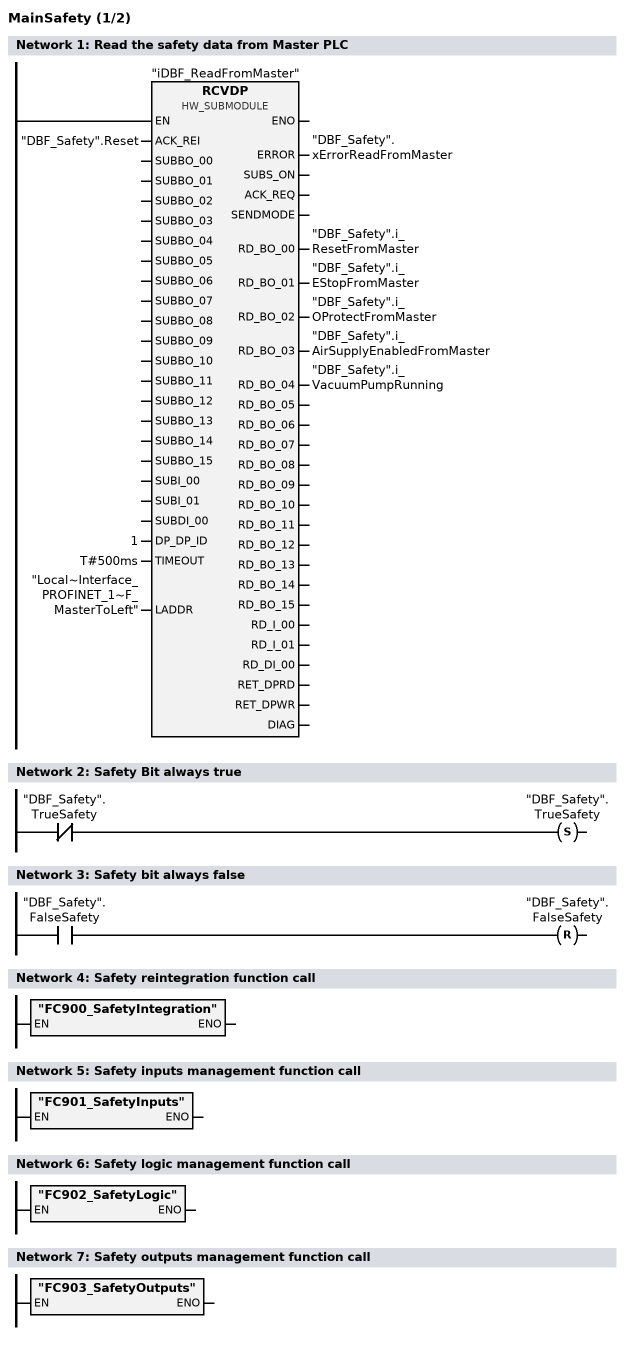
   RUNG wire#powerrail
      { S7_Templates := "laddr_type := HW_SUBMODULE" } "iDBF_ReadFromMaster".RCVDP(ACK_REI := "DBF_Safety".Reset, SUBBO_00 :=, SUBBO_01 :=, SUBBO_02 :=, SUBBO_03 :=, SUBBO_04 :=, SUBBO_05 :=, SUBBO_06 :=, SUBBO_07 :=, SUBBO_08 :=, SUBBO_09 :=, SUBBO_10 :=, SUBBO_11 :=, SUBBO_12 :=, SUBBO_13 :=, SUBBO_14 :=, SUBBO_15 :=, SUBI_00 :=, SUBI_01 :=, SUBDI_00 :=, DP_DP_ID := 1, TIMEOUT := T#500ms, LADDR := "Local~Interface_PROFINET_1~F_MasterToLeft", ERROR => "DBF_Safety".xErrorReadFromMaster, SUBS_ON =>, ACK_REQ =>, SENDMODE =>, RD_BO_00 => "DBF_Safety".i_ResetFromMaster, RD_BO_01 => "DBF_Safety".i_EStopFromMaster, RD_BO_02 => "DBF_Safety".i_OProtectFromMaster, RD_BO_03 => "DBF_Safety".i_AirSupplyEnabledFromMaster, RD_BO_04 => "DBF_Safety".i_VacuumPumpRunning, RD_BO_05 =>, RD_BO_06 =>, RD_BO_07 =>, RD_BO_08 =>, RD_BO_09 =>, RD_BO_10 =>, RD_BO_11 =>, RD_BO_12 =>, RD_BO_13 =>, RD_BO_14 =>, RD_BO_15 =>, RD_I_00 =>, RD_I_01 =>, RD_DI_00 =>, RET_DPRD =>, RET_DPWR =>, DIAG =>)
   END_RUNG
   // the same network as SCL:
   "iDBF_ReadFromMaster"(ACK_REI := "DBF_Safety".Reset,   // RCVDP
                         DP_DP_ID := 1,
                         TIMEOUT := T#500ms,
                         LADDR := "Local~Interface_PROFINET_1~F_MasterToLeft",
                         ERROR => "DBF_Safety".xErrorReadFromMaster,
                         RD_BO_00 => "DBF_Safety".i_ResetFromMaster,
                         RD_BO_01 => "DBF_Safety".i_EStopFromMaster,
                         RD_BO_02 => "DBF_Safety".i_OProtectFromMaster,
                         RD_BO_03 => "DBF_Safety".i_AirSupplyEnabledFromMaster,
                         RD_BO_04 => "DBF_Safety".i_VacuumPumpRunning);
END_REGION

REGION Network 2: Safety Bit always true
   RUNG wire#powerrail
      I_Contact( "DBF_Safety".TrueSafety )
      S_Coil( "DBF_Safety".TrueSafety )
   END_RUNG
   // the same network as SCL:
   IF NOT "DBF_Safety".TrueSafety THEN "DBF_Safety".TrueSafety := TRUE; END_IF;
END_REGION

REGION Network 3: Safety bit always false
   RUNG wire#powerrail
      Contact( "DBF_Safety".FalseSafety )
      R_Coil( "DBF_Safety".FalseSafety )
   END_RUNG
   // the same network as SCL:
   IF "DBF_Safety".FalseSafety THEN "DBF_Safety".FalseSafety := FALSE; END_IF;
END_REGION

REGION Network 4: Safety reintegration function call
   RUNG wire#powerrail
      "FC900_SafetyIntegration"()
   END_RUNG
   // the same network as SCL:
   "FC900_SafetyIntegration"();
END_REGION

REGION Network 5: Safety inputs management function call
   RUNG wire#powerrail
      "FC901_SafetyInputs"()
   END_RUNG
   // the same network as SCL:
   "FC901_SafetyInputs"();
END_REGION

REGION Network 6: Safety logic management function call
   RUNG wire#powerrail
      "FC902_SafetyLogic"()
   END_RUNG
   // the same network as SCL:
   "FC902_SafetyLogic"();
END_REGION

REGION Network 7: Safety outputs management function call
   RUNG wire#powerrail
      "FC903_SafetyOutputs"()
   END_RUNG
   // the same network as SCL:
   "FC903_SafetyOutputs"();
END_REGION

REGION Network 8: Write the safety data to Master PLC
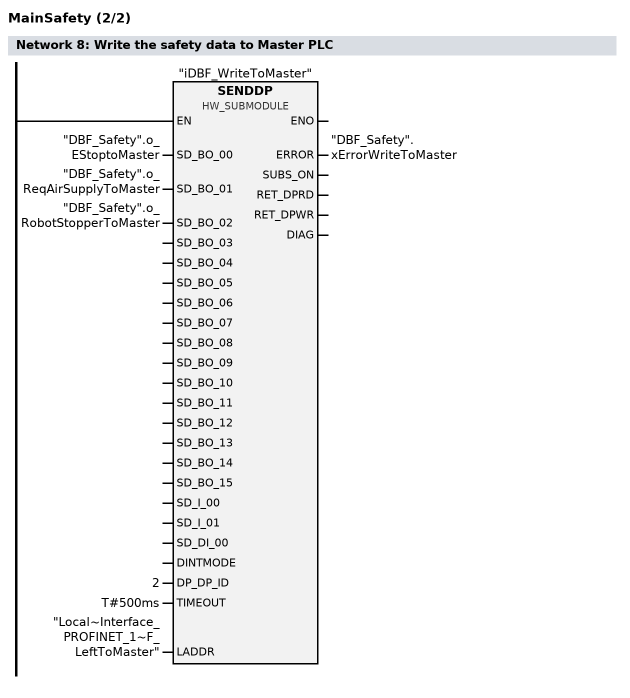
   RUNG wire#powerrail
      { S7_Templates := "laddr_type := HW_SUBMODULE" } "iDBF_WriteToMaster".SENDDP(SD_BO_00 := "DBF_Safety".o_EStoptoMaster, SD_BO_01 := "DBF_Safety".o_ReqAirSupplyToMaster, SD_BO_02 := "DBF_Safety".o_RobotStopperToMaster, SD_BO_03 :=, SD_BO_04 :=, SD_BO_05 :=, SD_BO_06 :=, SD_BO_07 :=, SD_BO_08 :=, SD_BO_09 :=, SD_BO_10 :=, SD_BO_11 :=, SD_BO_12 :=, SD_BO_13 :=, SD_BO_14 :=, SD_BO_15 :=, SD_I_00 :=, SD_I_01 :=, SD_DI_00 :=, DINTMODE :=, DP_DP_ID := 2, TIMEOUT := T#500ms, LADDR := "Local~Interface_PROFINET_1~F_LeftToMaster", ERROR => "DBF_Safety".xErrorWriteToMaster, SUBS_ON =>, RET_DPRD =>, RET_DPWR =>, DIAG =>)
   END_RUNG
   // the same network as SCL:
   "iDBF_WriteToMaster"(SD_BO_00 := "DBF_Safety".o_EStoptoMaster,   // SENDDP
                        SD_BO_01 := "DBF_Safety".o_ReqAirSupplyToMaster,
                        SD_BO_02 := "DBF_Safety".o_RobotStopperToMaster,
                        DP_DP_ID := 2,
                        TIMEOUT := T#500ms,
                        LADDR := "Local~Interface_PROFINET_1~F_LeftToMaster",
                        ERROR => "DBF_Safety".xErrorWriteToMaster);
END_REGION
END_FUNCTION_BLOCK

DATA_BLOCK "iDB_RobotComm"   // DB20
{ DB_Accessible_From_OPC_UA := 'FALSE' }
// stored: AutoNumber false, DBAccessibleFromOPCUA false, DBAccessibleFromWebserver false, InstanceOfName FB20 _RobotComm, InstanceOfType FB
"FB20 _RobotComm"
   // VAR_INPUT
   //    inCommRobot { ExternalAccessible := 'False'; ExternalVisible := 'False'; ExternalWritable := 'False'} : "stRecieveRobot";
   //    inCommMaster { ExternalAccessible := 'False'; ExternalVisible := 'False'; ExternalWritable := 'False'} : "stMasterToSlave";
   //    xEmergencyStop { ExternalAccessible := 'False'; ExternalVisible := 'False'; ExternalWritable := 'False'} : Bool;
   //    xOperatorProtection { ExternalAccessible := 'False'; ExternalVisible := 'False'; ExternalWritable := 'False'} : Bool;
   //    xResetFaultEStop { ExternalAccessible := 'False'; ExternalVisible := 'False'; ExternalWritable := 'False'} : Bool;
   //    xFaultPresent { ExternalAccessible := 'False'; ExternalVisible := 'False'; ExternalWritable := 'False'} : Bool;
   //    xFaultDiskRotation { ExternalAccessible := 'False'; ExternalVisible := 'False'; ExternalWritable := 'False'} : Bool;
   //    xAnalogSensorDetection { ExternalAccessible := 'False'; ExternalVisible := 'False'; ExternalWritable := 'False'} : Bool;
   //    rAnalogSensorValue { ExternalAccessible := 'False'; ExternalVisible := 'False'; ExternalWritable := 'False'} : Real;
   //    xVacuumValveClosed { ExternalAccessible := 'False'; ExternalVisible := 'False'; ExternalWritable := 'False'} : Bool;
   //    xVacuumValveOpen { ExternalAccessible := 'False'; ExternalVisible := 'False'; ExternalWritable := 'False'} : Bool;
   //    xDiskSensorLeft { ExternalAccessible := 'False'; ExternalVisible := 'False'; ExternalWritable := 'False'} : Bool;
   //    xDiskSensorRight { ExternalAccessible := 'False'; ExternalVisible := 'False'; ExternalWritable := 'False'} : Bool;
   //    xColorSensor1 { ExternalAccessible := 'False'; ExternalVisible := 'False'; ExternalWritable := 'False'} : Bool;
   //    xColorSensor2 { ExternalAccessible := 'False'; ExternalVisible := 'False'; ExternalWritable := 'False'} : Bool;
   //    xColorSensor3 { ExternalAccessible := 'False'; ExternalVisible := 'False'; ExternalWritable := 'False'} : Bool;
   //    xDiskTrayEmpty { ExternalAccessible := 'False'; ExternalVisible := 'False'; ExternalWritable := 'False'} : Bool;
   //    uiRobotSpeed { ExternalAccessible := 'False'; ExternalVisible := 'False'; ExternalWritable := 'False'} : UInt;
   //    xSandingReady { ExternalAccessible := 'False'; ExternalVisible := 'False'; ExternalWritable := 'False'} : Bool;
   //    xSandingDiskRotate { ExternalAccessible := 'False'; ExternalVisible := 'False'; ExternalWritable := 'False'} : Bool;
   //    xRemoveReady { ExternalAccessible := 'False'; ExternalVisible := 'False'; ExternalWritable := 'False'} : Bool;
   //    xPickUpReady { ExternalAccessible := 'False'; ExternalVisible := 'False'; ExternalWritable := 'False'} : Bool;
   //    xFlatnessCtrlReady { ExternalAccessible := 'False'; ExternalVisible := 'False'; ExternalWritable := 'False'} : Bool;
   //    xPulse { ExternalAccessible := 'False'; ExternalVisible := 'False'; ExternalWritable := 'False'} : Bool;
   //    uiWornPaperDistance { ExternalAccessible := 'False'; ExternalVisible := 'False'; ExternalWritable := 'False'} : UInt;
   //    rStrokePosition { ExternalAccessible := 'False'; ExternalVisible := 'False'; ExternalWritable := 'False'} : Real;
   //    rFlatnessPos { ExternalAccessible := 'False'; ExternalVisible := 'False'; ExternalWritable := 'False'} : Real;
   //    rDelta { ExternalAccessible := 'False'; ExternalVisible := 'False'; ExternalWritable := 'False'} : Real;
   //    usiNbDiskLeft { ExternalAccessible := 'False'; ExternalVisible := 'False'; ExternalWritable := 'False'} : USInt;
   //    usiNbDiskRight { ExternalAccessible := 'False'; ExternalVisible := 'False'; ExternalWritable := 'False'} : USInt;
   // END_VAR
   // VAR_OUTPUT
   //    outCommRobot { ExternalAccessible := 'False'; ExternalVisible := 'False'; ExternalWritable := 'False'} : "stSendRobot";
   //    xCleaningSensor { ExternalAccessible := 'False'; ExternalVisible := 'False'; ExternalWritable := 'False'} : Bool;
   //    xExecuteSanding { ExternalAccessible := 'False'; ExternalVisible := 'False'; ExternalWritable := 'False'} : Bool;
   //    xExecutePickUp { ExternalAccessible := 'False'; ExternalVisible := 'False'; ExternalWritable := 'False'} : Bool;
   //    xExecuteRemove { ExternalAccessible := 'False'; ExternalVisible := 'False'; ExternalWritable := 'False'} : Bool;
   //    xExecuteFlatnessCtrl { ExternalAccessible := 'False'; ExternalVisible := 'False'; ExternalWritable := 'False'} : Bool;
   //    xCloseVacuumValve { ExternalAccessible := 'False'; ExternalVisible := 'False'; ExternalWritable := 'False'} : Bool;
   //    xOpenVacuumValve { ExternalAccessible := 'False'; ExternalVisible := 'False'; ExternalWritable := 'False'} : Bool;
   //    xEnableSandingRotation { ExternalAccessible := 'False'; ExternalVisible := 'False'; ExternalWritable := 'False'} : Bool;
   //    xRunning { ExternalAccessible := 'False'; ExternalVisible := 'False'; ExternalWritable := 'False'} : Bool;
   //    xPause { ExternalAccessible := 'False'; ExternalVisible := 'False'; ExternalWritable := 'False'} : Bool;
   //    xFault { ExternalAccessible := 'False'; ExternalVisible := 'False'; ExternalWritable := 'False'} : Bool;
   //    uiJobNum { ExternalAccessible := 'False'; ExternalVisible := 'False'; ExternalWritable := 'False'} : UInt;
   //    xCmdManuRemoveDisk { ExternalAccessible := 'False'; ExternalVisible := 'False'; ExternalWritable := 'False'} : Bool;
   //    xCmdManuPickUpDisk { ExternalAccessible := 'False'; ExternalVisible := 'False'; ExternalWritable := 'False'} : Bool;
   //    xCmdManuFlatnessCtrl { ExternalAccessible := 'False'; ExternalVisible := 'False'; ExternalWritable := 'False'} : Bool;
   // END_VAR
   // VAR_IN_OUT
   //    xNewDisk { ExternalAccessible := 'False'; ExternalVisible := 'False'; ExternalWritable := 'False'} : Bool;
   //    xForceRotate { ExternalAccessible := 'False'; ExternalVisible := 'False'; ExternalWritable := 'False'} : Bool;
   //    outCommMaster : "stSlaveToMaster";
   // END_VAR
   // VAR
   //    nStepStartRecipe { ExternalAccessible := 'False'; ExternalVisible := 'False'; ExternalWritable := 'False'} : Int;
   //    nStepStartPath { ExternalAccessible := 'False'; ExternalVisible := 'False'; ExternalWritable := 'False'} : Int;
   // END_VAR
   // VAR RETAIN
   //    nStepChangePaper { ExternalAccessible := 'False'; ExternalVisible := 'False'; ExternalWritable := 'False'} : Int;
   //    nStepRemoveDisk { ExternalAccessible := 'False'; ExternalVisible := 'False'; ExternalWritable := 'False'} : Int;
   //    nStepPickupDisk { ExternalAccessible := 'False'; ExternalVisible := 'False'; ExternalWritable := 'False'} : Int;
   //    nStepControlDisk { ExternalAccessible := 'False'; ExternalVisible := 'False'; ExternalWritable := 'False'} : Int;
   //    nStepOperatorControl { ExternalAccessible := 'False'; ExternalVisible := 'False'; ExternalWritable := 'False'} : Int;
   //    nStepFlatnessControl { ExternalAccessible := 'False'; ExternalVisible := 'False'; ExternalWritable := 'False'} : Int;
   // END_VAR
   // VAR
   //    susiTryingCounter { ExternalAccessible := 'False'; ExternalVisible := 'False'; ExternalWritable := 'False'} : USInt;
   //    susiCountLeftSensor { ExternalAccessible := 'False'; ExternalVisible := 'False'; ExternalWritable := 'False'} : USInt;
   //    susiCountRightSensor { ExternalAccessible := 'False'; ExternalVisible := 'False'; ExternalWritable := 'False'} : USInt;
   //    suiInJobNum { ExternalAccessible := 'False'; ExternalVisible := 'False'; ExternalWritable := 'False'} : UInt;
   //    suiOutJobNum { ExternalAccessible := 'False'; ExternalVisible := 'False'; ExternalWritable := 'False'} : UInt;
   //    suiInDistanceSandingDisk { ExternalAccessible := 'False'; ExternalVisible := 'False'; ExternalWritable := 'False'} : UInt;
   //    suiInFrameNum { ExternalAccessible := 'False'; ExternalVisible := 'False'; ExternalWritable := 'False'} : UInt;
   //    suiInRobStatus { ExternalAccessible := 'False'; ExternalVisible := 'False'; ExternalWritable := 'False'} : UInt;
   //    suiInToolNum { ExternalAccessible := 'False'; ExternalVisible := 'False'; ExternalWritable := 'False'} : UInt;
   //    suiInPathNum { ExternalAccessible := 'False'; ExternalVisible := 'False'; ExternalWritable := 'False'} : UInt;
   //    suiOutRobotSpeedJob { ExternalAccessible := 'False'; ExternalVisible := 'False'; ExternalWritable := 'False'} : UInt;
   //    suiOutPathNum { ExternalAccessible := 'False'; ExternalVisible := 'False'; ExternalWritable := 'False'} : UInt;
   //    suiOutPlcDefNum { ExternalAccessible := 'False'; ExternalVisible := 'False'; ExternalWritable := 'False'} : UInt;
   //    suiOutPlcStatus { ExternalAccessible := 'False'; ExternalVisible := 'False'; ExternalWritable := 'False'} : UInt;
   //    suiOutRepereNum { ExternalAccessible := 'False'; ExternalVisible := 'False'; ExternalWritable := 'False'} : UInt;
   //    sxReqChangePaper { ExternalAccessible := 'False'; ExternalVisible := 'False'; ExternalWritable := 'False'} : Bool;
   //    sxChangeDiskFinished { ExternalAccessible := 'False'; ExternalVisible := 'False'; ExternalWritable := 'False'} : Bool;
   //    sxFPChangePaper { ExternalAccessible := 'False'; ExternalVisible := 'False'; ExternalWritable := 'False'} : Bool;
   //    sxChangeDiskReq { ExternalAccessible := 'False'; ExternalVisible := 'False'; ExternalWritable := 'False'} : Bool;
   //    sxDisckAReccorded { ExternalAccessible := 'False'; ExternalVisible := 'False'; ExternalWritable := 'False'} : Bool;
   //    sxDisckBReccorded { ExternalAccessible := 'False'; ExternalVisible := 'False'; ExternalWritable := 'False'} : Bool;
   //    sxDisckCReccorded { ExternalAccessible := 'False'; ExternalVisible := 'False'; ExternalWritable := 'False'} : Bool;
   //    sxFlatnessDiskAOk { ExternalAccessible := 'False'; ExternalVisible := 'False'; ExternalWritable := 'False'} : Bool;
   //    sxFlatnessDiskBOk { ExternalAccessible := 'False'; ExternalVisible := 'False'; ExternalWritable := 'False'} : Bool;
   //    sxFlatnessDiskCOk { ExternalAccessible := 'False'; ExternalVisible := 'False'; ExternalWritable := 'False'} : Bool;
   //    sxGlobalSafety { ExternalAccessible := 'False'; ExternalVisible := 'False'; ExternalWritable := 'False'} : Bool;
   //    sFPLeftSensor { ExternalAccessible := 'False'; ExternalVisible := 'False'; ExternalWritable := 'False'} : Bool;
   //    sFPRightSensor { ExternalAccessible := 'False'; ExternalVisible := 'False'; ExternalWritable := 'False'} : Bool;
   //    sxFPChangeDiskFinished { ExternalAccessible := 'False'; ExternalVisible := 'False'; ExternalWritable := 'False'} : Bool;
   //    sxDefaultRobot { ExternalAccessible := 'False'; ExternalVisible := 'False'; ExternalWritable := 'False'} : Bool;
   //    sxReqStartAgain { ExternalAccessible := 'False'; ExternalVisible := 'False'; ExternalWritable := 'False'} : Bool;
   //    sxForceFaultStep { ExternalAccessible := 'False'; ExternalVisible := 'False'; ExternalWritable := 'False'} : Bool;
   //    miDB_WatchDogRobot { ExternalAccessible := 'False'; ExternalVisible := 'False'; ExternalWritable := 'False'; S7_SetPoint := 'True'} : "FB_WatchDog";
   //    miDB_FP_DiskSensorLeft { ExternalAccessible := 'False'; ExternalVisible := 'False'; ExternalWritable := 'False'; S7_SetPoint := 'True'} : F_TRIG;
   //    miDB_FP_DiskSensorRight { ExternalAccessible := 'False'; ExternalVisible := 'False'; ExternalWritable := 'False'; S7_SetPoint := 'True'} : F_TRIG;
   //    miDB_TofLeftSensorFilter { ExternalAccessible := 'False'; ExternalVisible := 'False'; ExternalWritable := 'False'; S7_SetPoint := 'True'} : TOF_TIME;
   //    miDB_TofRightSensorFilter { ExternalAccessible := 'False'; ExternalVisible := 'False'; ExternalWritable := 'False'; S7_SetPoint := 'True'} : TOF_TIME;
   //    miDB_TofStartRecipe { ExternalAccessible := 'False'; ExternalVisible := 'False'; ExternalWritable := 'False'; S7_SetPoint := 'True'} : TOF_TIME;
   //    miDB_TonSandingDiskRotate { ExternalAccessible := 'False'; ExternalVisible := 'False'; ExternalWritable := 'False'; S7_SetPoint := 'True'} : TON_TIME;
   //    miDB_TonChangeDisk { ExternalAccessible := 'False'; ExternalVisible := 'False'; ExternalWritable := 'False'; S7_SetPoint := 'True'} : TON_TIME;
   //    miDB_TonTimeoutFeedBackProgNum { ExternalAccessible := 'False'; ExternalVisible := 'False'; ExternalWritable := 'False'; S7_SetPoint := 'True'} : TON_TIME;
   //    miDB_TonTimeoutFeedBackLaterType { ExternalAccessible := 'False'; ExternalVisible := 'False'; ExternalWritable := 'False'; S7_SetPoint := 'True'} : TON_TIME;
   // END_VAR
BEGIN
END_DATA_BLOCK

DATA_BLOCK "iDB_VacuumValve"   // DB50
{ DB_Accessible_From_OPC_UA := 'FALSE' }
// stored: AutoNumber false, DBAccessibleFromOPCUA false, DBAccessibleFromWebserver false, InstanceOfName FB_Actuator, InstanceOfType FB
"FB_Actuator"
   // VAR_INPUT
   //    xGlobalSafety { ExternalAccessible := 'False'; ExternalVisible := 'False'; ExternalWritable := 'False'} : Bool;
   //    xAuto { ExternalAccessible := 'False'; ExternalVisible := 'False'; ExternalWritable := 'False'} : Bool;
   //    xReset { ExternalAccessible := 'False'; ExternalVisible := 'False'; ExternalWritable := 'False'} : Bool;
   //    xHoming { ExternalAccessible := 'False'; ExternalVisible := 'False'; ExternalWritable := 'False'} : Bool;
   //    xActionning { ExternalAccessible := 'False'; ExternalVisible := 'False'; ExternalWritable := 'False'} : Bool;
   //    xResetCmd { ExternalAccessible := 'False'; ExternalVisible := 'False'; ExternalWritable := 'False'} : Bool;
   //    xPxHome { ExternalAccessible := 'False'; ExternalVisible := 'False'; ExternalWritable := 'False'} : Bool;
   //    xPxAction { ExternalAccessible := 'False'; ExternalVisible := 'False'; ExternalWritable := 'False'} : Bool;
   // END_VAR
   // VAR_OUTPUT
   //    xInHomePos { ExternalAccessible := 'False'; ExternalVisible := 'False'; ExternalWritable := 'False'} : Bool;
   //    xInActionPos { ExternalAccessible := 'False'; ExternalVisible := 'False'; ExternalWritable := 'False'} : Bool;
   //    xCmdHoming { ExternalAccessible := 'False'; ExternalVisible := 'False'; ExternalWritable := 'False'} : Bool;
   //    xCmdActionning { ExternalAccessible := 'False'; ExternalVisible := 'False'; ExternalWritable := 'False'} : Bool;
   //    wFault { ExternalAccessible := 'False'; ExternalVisible := 'False'; ExternalWritable := 'False'} : Word;
   // END_VAR
   // VAR_IN_OUT
   //    xHomingManu { ExternalAccessible := 'False'; ExternalVisible := 'False'; ExternalWritable := 'False'} : Bool;
   //    xActionningManu { ExternalAccessible := 'False'; ExternalVisible := 'False'; ExternalWritable := 'False'} : Bool;
   //    xResetCmdManu { ExternalAccessible := 'False'; ExternalVisible := 'False'; ExternalWritable := 'False'} : Bool;
   //    stActuatorConfig : "stConfigActuator";
   // END_VAR
   // VAR
   //    sxControlHoming { ExternalAccessible := 'False'; ExternalVisible := 'False'; ExternalWritable := 'False'} : Bool;
   //    sxControlActionning { ExternalAccessible := 'False'; ExternalVisible := 'False'; ExternalWritable := 'False'} : Bool;
   //    sxMemHoming { ExternalAccessible := 'False'; ExternalVisible := 'False'; ExternalWritable := 'False'} : Bool;
   //    sxMemActionning { ExternalAccessible := 'False'; ExternalVisible := 'False'; ExternalWritable := 'False'} : Bool;
   //    sxMemMeasureAverageHome { ExternalAccessible := 'False'; ExternalVisible := 'False'; ExternalWritable := 'False'} : Bool;
   //    sxMemMeasureAverageAction { ExternalAccessible := 'False'; ExternalVisible := 'False'; ExternalWritable := 'False'} : Bool;
   //    sxNewMemTimeHome { ExternalAccessible := 'False'; ExternalVisible := 'False'; ExternalWritable := 'False'} : Bool;
   //    sxNewMemTimeAction { ExternalAccessible := 'False'; ExternalVisible := 'False'; ExternalWritable := 'False'} : Bool;
   //    suiNbMeasureHome { ExternalAccessible := 'False'; ExternalVisible := 'False'; ExternalWritable := 'False'} : UInt;
   //    suiNbMeasureAction { ExternalAccessible := 'False'; ExternalVisible := 'False'; ExternalWritable := 'False'} : UInt;
   //    suiCount { ExternalAccessible := 'False'; ExternalVisible := 'False'; ExternalWritable := 'False'} : UInt;
   //    stMemTimeHome { ExternalAccessible := 'False'; ExternalVisible := 'False'; ExternalWritable := 'False'} : Time;
   //    stMemTimeAction { ExternalAccessible := 'False'; ExternalVisible := 'False'; ExternalWritable := 'False'} : Time;
   //    satAverageHoming { ExternalAccessible := 'False'; ExternalVisible := 'False'; ExternalWritable := 'False'; S7_SetPoint := 'True'} : Array[0..10] of Time;
   //    satAverageActionning { ExternalAccessible := 'False'; ExternalVisible := 'False'; ExternalWritable := 'False'} : Array[0..10] of Time;
   //    miDB_TonEnableHomingCommand { ExternalAccessible := 'False'; ExternalVisible := 'False'; ExternalWritable := 'False'; S7_SetPoint := 'True'} : TON_TIME;
   //    miDB_TonEnableActionningCommand { ExternalAccessible := 'False'; ExternalVisible := 'False'; ExternalWritable := 'False'; S7_SetPoint := 'True'} : TON_TIME;
   //    miDB_TonSimulateHomePxSensor { ExternalAccessible := 'False'; ExternalVisible := 'False'; ExternalWritable := 'False'; S7_SetPoint := 'True'} : TON_TIME;
   //    miDB_TonFilterHomePxSensor { ExternalAccessible := 'False'; ExternalVisible := 'False'; ExternalWritable := 'False'; S7_SetPoint := 'True'} : TON_TIME;
   //    miDB_TonSimulateActionPxSensor { ExternalAccessible := 'False'; ExternalVisible := 'False'; ExternalWritable := 'False'; S7_SetPoint := 'True'} : TON_TIME;
   //    miDB_TonFilterActionPxSensor { ExternalAccessible := 'False'; ExternalVisible := 'False'; ExternalWritable := 'False'; S7_SetPoint := 'True'} : TON_TIME;
   //    miDB_TonTimeoutHomeSensor { ExternalAccessible := 'False'; ExternalVisible := 'False'; ExternalWritable := 'False'; S7_SetPoint := 'True'} : TON_TIME;
   //    miDB_TonTimeoutActionSensor { ExternalAccessible := 'False'; ExternalVisible := 'False'; ExternalWritable := 'False'; S7_SetPoint := 'True'} : TON_TIME;
   //    miDB_FpPxHome { ExternalAccessible := 'False'; ExternalVisible := 'False'; ExternalWritable := 'False'; S7_SetPoint := 'True'} : R_TRIG;
   //    miDB_FpPxAction { ExternalAccessible := 'False'; ExternalVisible := 'False'; ExternalWritable := 'False'; S7_SetPoint := 'True'} : R_TRIG;
   // END_VAR
BEGIN
END_DATA_BLOCK

DATA_BLOCK "iDB_ManageTowerLight"   // DB60
{ DB_Accessible_From_OPC_UA := 'FALSE' }
// stored: AutoNumber false, DBAccessibleFromOPCUA false, DBAccessibleFromWebserver false, InstanceOfName FB60_ManageTowerLight, InstanceOfType FB
"FB60_ManageTowerLight"
   // VAR_INPUT
   //    xLightTest { ExternalAccessible := 'False'; ExternalVisible := 'False'; ExternalWritable := 'False'} : Bool;
   //    xConditionReady { ExternalAccessible := 'False'; ExternalVisible := 'False'; ExternalWritable := 'False'} : Bool;
   //    xStartUpWarning { ExternalAccessible := 'False'; ExternalVisible := 'False'; ExternalWritable := 'False'} : Bool;
   //    xReqOpActon { ExternalAccessible := 'False'; ExternalVisible := 'False'; ExternalWritable := 'False'} : Bool;
   //    xFault { ExternalAccessible := 'False'; ExternalVisible := 'False'; ExternalWritable := 'False'} : Bool;
   //    xPulseSlow { ExternalAccessible := 'False'; ExternalVisible := 'False'; ExternalWritable := 'False'} : Bool;
   //    xPulseFast { ExternalAccessible := 'False'; ExternalVisible := 'False'; ExternalWritable := 'False'} : Bool;
   // END_VAR
   // VAR_OUTPUT
   //    xGreenLight { ExternalAccessible := 'False'; ExternalVisible := 'False'; ExternalWritable := 'False'} : Bool;
   //    xOrangeLight { ExternalAccessible := 'False'; ExternalVisible := 'False'; ExternalWritable := 'False'} : Bool;
   //    xRedLight { ExternalAccessible := 'False'; ExternalVisible := 'False'; ExternalWritable := 'False'} : Bool;
   //    xBuzzer { ExternalAccessible := 'False'; ExternalVisible := 'False'; ExternalWritable := 'False'} : Bool;
   // END_VAR
   // VAR
   //    miDB_TpNewFault { ExternalAccessible := 'False'; ExternalVisible := 'False'; ExternalWritable := 'False'; S7_SetPoint := 'True'} : TP_TIME;
   // END_VAR
BEGIN
END_DATA_BLOCK

DATA_BLOCK "iDB_CounterChangingDisk"   // DB73
{ S7_Optimized_Access := 'TRUE'; DB_Accessible_From_OPC_UA := 'FALSE' }
// stored: AutoNumber false, DBAccessibleFromOPCUA false, DBAccessibleFromWebserver false, InstanceOfName IEC_UCOUNTER, OfSystemLibElement IEC_UCOUNTER, OfSystemLibVersion 1.0
"IEC_UCOUNTER"
   // VAR RETAIN
   //    CU : Bool;
   //    CD : Bool;
   //    R : Bool;
   //    LD : Bool;
   //    QU : Bool;
   //    QD : Bool;
   //    PV : UInt;
   //    CV : UInt;
   // END_VAR
BEGIN
END_DATA_BLOCK

DATA_BLOCK "iDB_RobotDriveOnCounter"   // DB75
// stored: AutoNumber false, InstanceOfName FB_TimeCounter, InstanceOfType FB
"FB_TimeCounter"
   // VAR_INPUT
   //    xClockSecond { ExternalAccessible := 'False'; ExternalVisible := 'False'; ExternalWritable := 'False'} : Bool;
   //    xStart { ExternalAccessible := 'False'; ExternalVisible := 'False'; ExternalWritable := 'False'} : Bool;
   //    xStop { ExternalAccessible := 'False'; ExternalVisible := 'False'; ExternalWritable := 'False'} : Bool;
   //    xResetCounter { ExternalAccessible := 'False'; ExternalVisible := 'False'; ExternalWritable := 'False'} : Bool;
   // END_VAR
   // VAR_OUTPUT
   //    PerpetualCounter { ExternalAccessible := 'False'; ExternalVisible := 'False'; ExternalWritable := 'False'} : UDInt;
   //    "Counter" { ExternalAccessible := 'False'; ExternalVisible := 'False'; ExternalWritable := 'False'} : UDInt;
   // END_VAR
   // VAR
   //    sxEnableCount { ExternalAccessible := 'False'; ExternalVisible := 'False'; ExternalWritable := 'False'} : Bool;
   //    sxFpStart { ExternalAccessible := 'False'; ExternalVisible := 'False'; ExternalWritable := 'False'} : Bool;
   //    sxFpStop { ExternalAccessible := 'False'; ExternalVisible := 'False'; ExternalWritable := 'False'} : Bool;
   // END_VAR
   // VAR RETAIN
   //    miDB_Counter { ExternalAccessible := 'False'; ExternalVisible := 'False'; ExternalWritable := 'False'; S7_SetPoint := 'True'} : CTU_UDINT;
   //    miDB_PerpetualCount { ExternalAccessible := 'False'; ExternalVisible := 'False'; ExternalWritable := 'False'; S7_SetPoint := 'True'} : CTU_UDINT;
   // END_VAR
   // VAR
   //    sxFpResetCounter { ExternalAccessible := 'False'; ExternalVisible := 'False'; ExternalWritable := 'False'} : Bool;
   //    sxResetCounter { ExternalAccessible := 'False'; ExternalVisible := 'False'; ExternalWritable := 'False'} : Bool;
   // END_VAR
BEGIN
END_DATA_BLOCK

DATA_BLOCK "iDB_RobotPowerOnCounter"   // DB74
// stored: AutoNumber false, InstanceOfName FB_TimeCounter, InstanceOfType FB
"FB_TimeCounter"
   // VAR_INPUT
   //    xClockSecond { ExternalAccessible := 'False'; ExternalVisible := 'False'; ExternalWritable := 'False'} : Bool;
   //    xStart { ExternalAccessible := 'False'; ExternalVisible := 'False'; ExternalWritable := 'False'} : Bool;
   //    xStop { ExternalAccessible := 'False'; ExternalVisible := 'False'; ExternalWritable := 'False'} : Bool;
   //    xResetCounter { ExternalAccessible := 'False'; ExternalVisible := 'False'; ExternalWritable := 'False'} : Bool;
   // END_VAR
   // VAR_OUTPUT
   //    PerpetualCounter { ExternalAccessible := 'False'; ExternalVisible := 'False'; ExternalWritable := 'False'} : UDInt;
   //    "Counter" { ExternalAccessible := 'False'; ExternalVisible := 'False'; ExternalWritable := 'False'} : UDInt;
   // END_VAR
   // VAR
   //    sxEnableCount { ExternalAccessible := 'False'; ExternalVisible := 'False'; ExternalWritable := 'False'} : Bool;
   //    sxFpStart { ExternalAccessible := 'False'; ExternalVisible := 'False'; ExternalWritable := 'False'} : Bool;
   //    sxFpStop { ExternalAccessible := 'False'; ExternalVisible := 'False'; ExternalWritable := 'False'} : Bool;
   // END_VAR
   // VAR RETAIN
   //    miDB_Counter { ExternalAccessible := 'False'; ExternalVisible := 'False'; ExternalWritable := 'False'; S7_SetPoint := 'True'} : CTU_UDINT;
   //    miDB_PerpetualCount { ExternalAccessible := 'False'; ExternalVisible := 'False'; ExternalWritable := 'False'; S7_SetPoint := 'True'} : CTU_UDINT;
   // END_VAR
   // VAR
   //    sxFpResetCounter { ExternalAccessible := 'False'; ExternalVisible := 'False'; ExternalWritable := 'False'} : Bool;
   //    sxResetCounter { ExternalAccessible := 'False'; ExternalVisible := 'False'; ExternalWritable := 'False'} : Bool;
   // END_VAR
BEGIN
END_DATA_BLOCK

DATA_BLOCK "iDB_TimeCounterFault"   // DB72
{ DB_Accessible_From_OPC_UA := 'FALSE' }
// stored: AutoNumber false, DBAccessibleFromOPCUA false, DBAccessibleFromWebserver false, InstanceOfName FB_TimeCounter, InstanceOfType FB
"FB_TimeCounter"
   // VAR_INPUT
   //    xClockSecond { ExternalAccessible := 'False'; ExternalVisible := 'False'; ExternalWritable := 'False'} : Bool;
   //    xStart { ExternalAccessible := 'False'; ExternalVisible := 'False'; ExternalWritable := 'False'} : Bool;
   //    xStop { ExternalAccessible := 'False'; ExternalVisible := 'False'; ExternalWritable := 'False'} : Bool;
   //    xResetCounter { ExternalAccessible := 'False'; ExternalVisible := 'False'; ExternalWritable := 'False'} : Bool;
   // END_VAR
   // VAR_OUTPUT
   //    PerpetualCounter { ExternalAccessible := 'False'; ExternalVisible := 'False'; ExternalWritable := 'False'} : UDInt;
   //    "Counter" { ExternalAccessible := 'False'; ExternalVisible := 'False'; ExternalWritable := 'False'} : UDInt;
   // END_VAR
   // VAR
   //    sxEnableCount { ExternalAccessible := 'False'; ExternalVisible := 'False'; ExternalWritable := 'False'} : Bool;
   //    sxFpStart { ExternalAccessible := 'False'; ExternalVisible := 'False'; ExternalWritable := 'False'} : Bool;
   //    sxFpStop { ExternalAccessible := 'False'; ExternalVisible := 'False'; ExternalWritable := 'False'} : Bool;
   // END_VAR
   // VAR RETAIN
   //    miDB_Counter { ExternalAccessible := 'False'; ExternalVisible := 'False'; ExternalWritable := 'False'; S7_SetPoint := 'True'} : CTU_UDINT;
   //    miDB_PerpetualCount { ExternalAccessible := 'False'; ExternalVisible := 'False'; ExternalWritable := 'False'; S7_SetPoint := 'True'} : CTU_UDINT;
   // END_VAR
   // VAR
   //    sxFpResetCounter { ExternalAccessible := 'False'; ExternalVisible := 'False'; ExternalWritable := 'False'} : Bool;
   //    sxResetCounter { ExternalAccessible := 'False'; ExternalVisible := 'False'; ExternalWritable := 'False'} : Bool;
   // END_VAR
BEGIN
END_DATA_BLOCK

DATA_BLOCK "iDB_TimeCounterRunning"   // DB70
{ DB_Accessible_From_OPC_UA := 'FALSE' }
// stored: AutoNumber false, DBAccessibleFromOPCUA false, DBAccessibleFromWebserver false, InstanceOfName FB_TimeCounter, InstanceOfType FB
"FB_TimeCounter"
   // VAR_INPUT
   //    xClockSecond { ExternalAccessible := 'False'; ExternalVisible := 'False'; ExternalWritable := 'False'} : Bool;
   //    xStart { ExternalAccessible := 'False'; ExternalVisible := 'False'; ExternalWritable := 'False'} : Bool;
   //    xStop { ExternalAccessible := 'False'; ExternalVisible := 'False'; ExternalWritable := 'False'} : Bool;
   //    xResetCounter { ExternalAccessible := 'False'; ExternalVisible := 'False'; ExternalWritable := 'False'} : Bool;
   // END_VAR
   // VAR_OUTPUT
   //    PerpetualCounter { ExternalAccessible := 'False'; ExternalVisible := 'False'; ExternalWritable := 'False'} : UDInt;
   //    "Counter" { ExternalAccessible := 'False'; ExternalVisible := 'False'; ExternalWritable := 'False'} : UDInt;
   // END_VAR
   // VAR
   //    sxEnableCount { ExternalAccessible := 'False'; ExternalVisible := 'False'; ExternalWritable := 'False'} : Bool;
   //    sxFpStart { ExternalAccessible := 'False'; ExternalVisible := 'False'; ExternalWritable := 'False'} : Bool;
   //    sxFpStop { ExternalAccessible := 'False'; ExternalVisible := 'False'; ExternalWritable := 'False'} : Bool;
   // END_VAR
   // VAR RETAIN
   //    miDB_Counter { ExternalAccessible := 'False'; ExternalVisible := 'False'; ExternalWritable := 'False'; S7_SetPoint := 'True'} : CTU_UDINT;
   //    miDB_PerpetualCount { ExternalAccessible := 'False'; ExternalVisible := 'False'; ExternalWritable := 'False'; S7_SetPoint := 'True'} : CTU_UDINT;
   // END_VAR
   // VAR
   //    sxFpResetCounter { ExternalAccessible := 'False'; ExternalVisible := 'False'; ExternalWritable := 'False'} : Bool;
   //    sxResetCounter { ExternalAccessible := 'False'; ExternalVisible := 'False'; ExternalWritable := 'False'} : Bool;
   // END_VAR
BEGIN
END_DATA_BLOCK

DATA_BLOCK "iDB_GreasingZAxis"   // DB80
// stored: AutoNumber false, InstanceOfName FB80_Greasing, InstanceOfType FB
"FB80_Greasing"
   // VAR_INPUT
   //    xForcingGreasing { ExternalAccessible := 'False'; ExternalVisible := 'False'; ExternalWritable := 'False'} : Bool;
   //    xResetGreasingFault { ExternalAccessible := 'False'; ExternalVisible := 'False'; ExternalWritable := 'False'} : Bool;
   //    xPxPignon { ExternalAccessible := 'False'; ExternalVisible := 'False'; ExternalWritable := 'False'} : Bool;
   //    xPxGrease { ExternalAccessible := 'False'; ExternalVisible := 'False'; ExternalWritable := 'False'} : Bool;
   //    Config { ExternalAccessible := 'False'; ExternalVisible := 'False'; ExternalWritable := 'False'} : "stConfigGrease";
   // END_VAR
   // VAR_OUTPUT
   //    xGreaseProgRunning { ExternalAccessible := 'False'; ExternalVisible := 'False'; ExternalWritable := 'False'} : Bool;
   //    xGreaseFault { ExternalAccessible := 'False'; ExternalVisible := 'False'; ExternalWritable := 'False'} : Bool;
   //    xEnableGreasePumpe { ExternalAccessible := 'False'; ExternalVisible := 'False'; ExternalWritable := 'False'} : Bool;
   //    uiCounterPulse { ExternalAccessible := 'False'; ExternalVisible := 'False'; ExternalWritable := 'False'} : UInt;
   //    uiGreaseFault { ExternalAccessible := 'False'; ExternalVisible := 'False'; ExternalWritable := 'False'} : UInt;
   //    udiTotalOdometer { ExternalAccessible := 'False'; ExternalVisible := 'False'; ExternalWritable := 'False'} : UDInt;
   //    uiCurrOdometer : UInt;
   // END_VAR
   // VAR RETAIN
   //    miDB_CtPignonPxSensor { ExternalAccessible := 'False'; ExternalVisible := 'False'; ExternalWritable := 'False'; S7_SetPoint := 'True'} : CTU_UINT;
   //    miDB_CtOdometer { ExternalAccessible := 'False'; ExternalVisible := 'False'; ExternalWritable := 'False'; S7_SetPoint := 'True'} : CTU_UINT;
   //    miDB_CtGreaseFault { ExternalAccessible := 'False'; ExternalVisible := 'False'; ExternalWritable := 'False'; S7_SetPoint := 'True'} : CTU_UINT;
   //    miDB_CtRestartCycle { ExternalAccessible := 'False'; ExternalVisible := 'False'; ExternalWritable := 'False'; S7_SetPoint := 'True'} : CTU_INT;
   //    miDB_CtOdometerTotalizater { ExternalAccessible := 'False'; ExternalVisible := 'False'; ExternalWritable := 'False'; S7_SetPoint := 'True'} : CTU_UDINT;
   // END_VAR
   // VAR
   //    miDB_TonEndCtrlGreasePx { ExternalAccessible := 'False'; ExternalVisible := 'False'; ExternalWritable := 'False'; S7_SetPoint := 'True'} : TON_TIME;
   //    miDB_TpActivePump { ExternalAccessible := 'False'; ExternalVisible := 'False'; ExternalWritable := 'False'; S7_SetPoint := 'True'} : TP_TIME;
   //    miDB_TpGreaseFaultActive { ExternalAccessible := 'False'; ExternalVisible := 'False'; ExternalWritable := 'False'; S7_SetPoint := 'True'} : TP_TIME;
   //    miDB_TsspCtrlGreasePx { ExternalAccessible := 'False'; ExternalVisible := 'False'; ExternalWritable := 'False'; S7_SetPoint := 'True'} : "FB_TSSP";
   //    miDB_TsspCtrlMove { ExternalAccessible := 'False'; ExternalVisible := 'False'; ExternalWritable := 'False'; S7_SetPoint := 'True'} : "FB_TSSP";
   //    sxOneKm { ExternalAccessible := 'False'; ExternalVisible := 'False'; ExternalWritable := 'False'} : Bool;
   //    sxOdometer { ExternalAccessible := 'False'; ExternalVisible := 'False'; ExternalWritable := 'False'} : Bool;
   //    xResetCtPignonPxSensor { ExternalAccessible := 'False'; ExternalVisible := 'False'; ExternalWritable := 'False'} : Bool;
   //    sxResetCtOdomoter { ExternalAccessible := 'False'; ExternalVisible := 'False'; ExternalWritable := 'False'} : Bool;
   //    sxResetCtRestartCycle { ExternalAccessible := 'False'; ExternalVisible := 'False'; ExternalWritable := 'False'} : Bool;
   //    sxMemActivationGreasePump { ExternalAccessible := 'False'; ExternalVisible := 'False'; ExternalWritable := 'False'} : Bool;
   //    sxMemOffGreasePx { ExternalAccessible := 'False'; ExternalVisible := 'False'; ExternalWritable := 'False'} : Bool;
   //    sxMemOnGreasePx { ExternalAccessible := 'False'; ExternalVisible := 'False'; ExternalWritable := 'False'} : Bool;
   //    sxFPEnableGreasePumpe { ExternalAccessible := 'False'; ExternalVisible := 'False'; ExternalWritable := 'False'} : Bool;
   // END_VAR
BEGIN
END_DATA_BLOCK

DATA_BLOCK "iDBF_ExternalEStopToRobot"   // DB942, F_DB
{ DB_Accessible_From_OPC_UA := 'FALSE' }
// stored: AutoNumber false, DBAccessibleFromOPCUA false, DBAccessibleFromWebserver false, InstanceOfName SafetyOutputControled, InstanceOfType FB
"SafetyOutputControled"
   // VAR_INPUT
   //    xControlSafety { ExternalAccessible := 'False'; ExternalVisible := 'False'; ExternalWritable := 'False'} : Bool;
   //    xInputFdb { ExternalAccessible := 'False'; ExternalVisible := 'False'; ExternalWritable := 'False'} : Bool;
   //    xOutputState { ExternalAccessible := 'False'; ExternalVisible := 'False'; ExternalWritable := 'False'} : Bool;
   //    tFdbTime { ExternalAccessible := 'False'; ExternalVisible := 'False'; ExternalWritable := 'False'} : Time;
   //    xAck { ExternalAccessible := 'False'; ExternalVisible := 'False'; ExternalWritable := 'False'} : Bool;
   //    xAllowAck { ExternalAccessible := 'False'; ExternalVisible := 'False'; ExternalWritable := 'False'} : Bool;
   // END_VAR
   // VAR_OUTPUT
   //    xOutputSafety { ExternalAccessible := 'False'; ExternalVisible := 'False'; ExternalWritable := 'False'} : Bool;
   //    stSafetyState { ExternalAccessible := 'False'; ExternalVisible := 'False'; ExternalWritable := 'False'} : "stSafetyState";
   // END_VAR
   // VAR
   //    miDBF_OutFeedBack { ExternalAccessible := 'False'; ExternalVisible := 'False'; ExternalWritable := 'False'} : FDBACK;
   //    sx_Ack { ExternalAccessible := 'False'; ExternalVisible := 'False'; ExternalWritable := 'False'} : Bool;
   //    sx_TempAck { ExternalAccessible := 'False'; ExternalVisible := 'False'; ExternalWritable := 'False'} : Bool;
   //    sx_TempAckReq { ExternalAccessible := 'False'; ExternalVisible := 'False'; ExternalWritable := 'False'} : Bool;
   //    sx_TempError { ExternalAccessible := 'False'; ExternalVisible := 'False'; ExternalWritable := 'False'} : Bool;
   // END_VAR
BEGIN
END_DATA_BLOCK

DATA_BLOCK "iDBF_ExternalOProtectToRobot"   // DB953, F_DB
{ DB_Accessible_From_OPC_UA := 'FALSE' }
// stored: AutoNumber false, DBAccessibleFromOPCUA false, DBAccessibleFromWebserver false, InstanceOfName SafetyOutputControled, InstanceOfType FB
"SafetyOutputControled"
   // VAR_INPUT
   //    xControlSafety { ExternalAccessible := 'False'; ExternalVisible := 'False'; ExternalWritable := 'False'} : Bool;
   //    xInputFdb { ExternalAccessible := 'False'; ExternalVisible := 'False'; ExternalWritable := 'False'} : Bool;
   //    xOutputState { ExternalAccessible := 'False'; ExternalVisible := 'False'; ExternalWritable := 'False'} : Bool;
   //    tFdbTime { ExternalAccessible := 'False'; ExternalVisible := 'False'; ExternalWritable := 'False'} : Time;
   //    xAck { ExternalAccessible := 'False'; ExternalVisible := 'False'; ExternalWritable := 'False'} : Bool;
   //    xAllowAck { ExternalAccessible := 'False'; ExternalVisible := 'False'; ExternalWritable := 'False'} : Bool;
   // END_VAR
   // VAR_OUTPUT
   //    xOutputSafety { ExternalAccessible := 'False'; ExternalVisible := 'False'; ExternalWritable := 'False'} : Bool;
   //    stSafetyState { ExternalAccessible := 'False'; ExternalVisible := 'False'; ExternalWritable := 'False'} : "stSafetyState";
   // END_VAR
   // VAR
   //    miDBF_OutFeedBack { ExternalAccessible := 'False'; ExternalVisible := 'False'; ExternalWritable := 'False'} : FDBACK;
   //    sx_Ack { ExternalAccessible := 'False'; ExternalVisible := 'False'; ExternalWritable := 'False'} : Bool;
   //    sx_TempAck { ExternalAccessible := 'False'; ExternalVisible := 'False'; ExternalWritable := 'False'} : Bool;
   //    sx_TempAckReq { ExternalAccessible := 'False'; ExternalVisible := 'False'; ExternalWritable := 'False'} : Bool;
   //    sx_TempError { ExternalAccessible := 'False'; ExternalVisible := 'False'; ExternalWritable := 'False'} : Bool;
   // END_VAR
BEGIN
END_DATA_BLOCK

DATA_BLOCK "iDBF_OpenZAxisBrake"   // DB940, F_DB
{ DB_Accessible_From_OPC_UA := 'FALSE' }
// stored: AutoNumber false, DBAccessibleFromOPCUA false, DBAccessibleFromWebserver false, InstanceOfName SafetyOutputControled, InstanceOfType FB
"SafetyOutputControled"
   // VAR_INPUT
   //    xControlSafety { ExternalAccessible := 'False'; ExternalVisible := 'False'; ExternalWritable := 'False'} : Bool;
   //    xInputFdb { ExternalAccessible := 'False'; ExternalVisible := 'False'; ExternalWritable := 'False'} : Bool;
   //    xOutputState { ExternalAccessible := 'False'; ExternalVisible := 'False'; ExternalWritable := 'False'} : Bool;
   //    tFdbTime { ExternalAccessible := 'False'; ExternalVisible := 'False'; ExternalWritable := 'False'} : Time;
   //    xAck { ExternalAccessible := 'False'; ExternalVisible := 'False'; ExternalWritable := 'False'} : Bool;
   //    xAllowAck { ExternalAccessible := 'False'; ExternalVisible := 'False'; ExternalWritable := 'False'} : Bool;
   // END_VAR
   // VAR_OUTPUT
   //    xOutputSafety { ExternalAccessible := 'False'; ExternalVisible := 'False'; ExternalWritable := 'False'} : Bool;
   //    stSafetyState { ExternalAccessible := 'False'; ExternalVisible := 'False'; ExternalWritable := 'False'} : "stSafetyState";
   // END_VAR
   // VAR
   //    miDBF_OutFeedBack { ExternalAccessible := 'False'; ExternalVisible := 'False'; ExternalWritable := 'False'} : FDBACK;
   //    sx_Ack { ExternalAccessible := 'False'; ExternalVisible := 'False'; ExternalWritable := 'False'} : Bool;
   //    sx_TempAck { ExternalAccessible := 'False'; ExternalVisible := 'False'; ExternalWritable := 'False'} : Bool;
   //    sx_TempAckReq { ExternalAccessible := 'False'; ExternalVisible := 'False'; ExternalWritable := 'False'} : Bool;
   //    sx_TempError { ExternalAccessible := 'False'; ExternalVisible := 'False'; ExternalWritable := 'False'} : Bool;
   // END_VAR
BEGIN
END_DATA_BLOCK

DATA_BLOCK "iDBF_PowerOffFerRobotic"   // DB943, F_DB
{ DB_Accessible_From_OPC_UA := 'FALSE' }
// stored: AutoNumber false, DBAccessibleFromOPCUA false, DBAccessibleFromWebserver false, InstanceOfName SafetyOutputControled, InstanceOfType FB
"SafetyOutputControled"
   // VAR_INPUT
   //    xControlSafety { ExternalAccessible := 'False'; ExternalVisible := 'False'; ExternalWritable := 'False'} : Bool;
   //    xInputFdb { ExternalAccessible := 'False'; ExternalVisible := 'False'; ExternalWritable := 'False'} : Bool;
   //    xOutputState { ExternalAccessible := 'False'; ExternalVisible := 'False'; ExternalWritable := 'False'} : Bool;
   //    tFdbTime { ExternalAccessible := 'False'; ExternalVisible := 'False'; ExternalWritable := 'False'} : Time;
   //    xAck { ExternalAccessible := 'False'; ExternalVisible := 'False'; ExternalWritable := 'False'} : Bool;
   //    xAllowAck { ExternalAccessible := 'False'; ExternalVisible := 'False'; ExternalWritable := 'False'} : Bool;
   // END_VAR
   // VAR_OUTPUT
   //    xOutputSafety { ExternalAccessible := 'False'; ExternalVisible := 'False'; ExternalWritable := 'False'} : Bool;
   //    stSafetyState { ExternalAccessible := 'False'; ExternalVisible := 'False'; ExternalWritable := 'False'} : "stSafetyState";
   // END_VAR
   // VAR
   //    miDBF_OutFeedBack { ExternalAccessible := 'False'; ExternalVisible := 'False'; ExternalWritable := 'False'} : FDBACK;
   //    sx_Ack { ExternalAccessible := 'False'; ExternalVisible := 'False'; ExternalWritable := 'False'} : Bool;
   //    sx_TempAck { ExternalAccessible := 'False'; ExternalVisible := 'False'; ExternalWritable := 'False'} : Bool;
   //    sx_TempAckReq { ExternalAccessible := 'False'; ExternalVisible := 'False'; ExternalWritable := 'False'} : Bool;
   //    sx_TempError { ExternalAccessible := 'False'; ExternalVisible := 'False'; ExternalWritable := 'False'} : Bool;
   // END_VAR
BEGIN
END_DATA_BLOCK

DATA_BLOCK "iDBF_StopStrokeLimit"   // DB944, F_DB
{ DB_Accessible_From_OPC_UA := 'FALSE' }
// stored: AutoNumber false, DBAccessibleFromOPCUA false, DBAccessibleFromWebserver false, InstanceOfName EmergencyStop, InstanceOfType FB
"EmergencyStop"
   // VAR_INPUT
   //    xInputSafety { ExternalAccessible := 'False'; ExternalVisible := 'False'; ExternalWritable := 'False'} : Bool;
   //    xStateInput { ExternalAccessible := 'False'; ExternalVisible := 'False'; ExternalWritable := 'False'} : Bool;
   //    xAck { ExternalAccessible := 'False'; ExternalVisible := 'False'; ExternalWritable := 'False'} : Bool;
   //    xAllowAck { ExternalAccessible := 'False'; ExternalVisible := 'False'; ExternalWritable := 'False'} : Bool;
   // END_VAR
   // VAR_OUTPUT
   //    xStateSafety { ExternalAccessible := 'False'; ExternalVisible := 'False'; ExternalWritable := 'False'} : Bool;
   //    stSafetyState { ExternalAccessible := 'False'; ExternalVisible := 'False'; ExternalWritable := 'False'} : "stSafetyState";
   // END_VAR
   // VAR
   //    sx_Ack { ExternalAccessible := 'False'; ExternalVisible := 'False'; ExternalWritable := 'False'} : Bool;
   //    sx_TempAck { ExternalAccessible := 'False'; ExternalVisible := 'False'; ExternalWritable := 'False'} : Bool;
   //    sx_TempAckReq { ExternalAccessible := 'False'; ExternalVisible := 'False'; ExternalWritable := 'False'} : Bool;
   //    miDBF_EStop { ExternalAccessible := 'False'; ExternalVisible := 'False'; ExternalWritable := 'False'} : ESTOP1;
   // END_VAR
BEGIN
END_DATA_BLOCK
